LIN {X 0,Y 445.491,Z 467.925,A -85,B 0,C 180,E1 -8723.659,E2 -8723.659} C_VEL
LIN {X 0,Y 445.471,Z 472.126,A -85,B 0,C 180,E1 -8725.021,E2 -8725.021} C_VEL
LIN {X 0,Y 445.391,Z 475.228,A -85,B 0,C 180,E1 -8726.38,E2 -8726.38} C_VEL
LIN {X 0,Y 445.448,Z 476.703,A -85,B 0,C 180,E1 -8727.286,E2 -8727.286} C_VEL
LIN {X 0,Y 445.399,Z 477.757,A -85,B 0,C 180,E1 -8728.191,E2 -8728.191} C_VEL
LIN {X 0,Y 445.398,Z 478.402,A -85,B 0,C 180,E1 -8729.095,E2 -8729.095} C_VEL
LIN {X 0,Y 445.406,Z 478.591,A -85,B 0,C 180,E1 -8729.999,E2 -8729.999} C_VEL
LIN {X 0,Y 445.398,Z 478.345,A -85,B 0,C 180,E1 -8730.903,E2 -8730.903} C_VEL
LIN {X 0,Y 445.399,Z 477.688,A -85,B 0,C 180,E1 -8731.807,E2 -8731.807} C_VEL
LIN {X 0,Y 445.452,Z 476.615,A -85,B 0,C 180,E1 -8732.712,E2 -8732.712} C_VEL
LIN {X 0,Y 445.399,Z 474.132,A -85,B 0,C 180,E1 -8734.071,E2 -8734.071} C_VEL
LIN {X 0,Y 445.479,Z 470.6,A -85,B 0,C 180,E1 -8735.431,E2 -8735.431} C_VEL
LIN {X 0,Y 445.542,Z 465.911,A -85,B 0,C 180,E1 -8736.793,E2 -8736.793} C_VEL
LIN {X 0,Y 445.738,Z 459.918,A -85,B 0,C 180,E1 -8738.157,E2 -8738.157} C_VEL
LIN {X 0,Y 446.06,Z 449.817,A -85,B 0,C 180,E1 -8739.979,E2 -8739.979} C_VEL
LIN {X 0,Y 446.499,Z 442.125,A -85,B 0,C 180,E1 -8741.116,E2 -8741.116} C_VEL
LIN {X 0,Y 447.018,Z 432.751,A -85,B 0,C 180,E1 -8742.253,E2 -8742.253} C_VEL
LIN {X 0,Y 447.601,Z 421.509,A -85,B 0,C 180,E1 -8743.348,E2 -8743.348} C_VEL
LIN {X 0,Y 448.216,Z 410.725,A -85,B 0,C 180,E1 -8744.181,E2 -8744.181} C_VEL
LIN {X 0,Y 448.805,Z 398.322,A -85,B 0,C 180,E1 -8744.915,E2 -8744.915} C_VEL
LIN {X 0,Y 449.352,Z 385.98,A -85,B 0,C 180,E1 -8745.448,E2 -8745.448} C_VEL
LIN {X 0,Y 449.771,Z 373.319,A -85,B 0,C 180,E1 -8745.81,E2 -8745.81} C_VEL
LIN {X 0,Y 450.349,Z 287.235,A -85,B 0,C 180,E1 -8747.236,E2 -8747.236} C_VEL
LIN {X 0,Y 447.336,Z 266.21,A -85,B 0,C 180,E1 -8747.733,E2 -8747.733} C_VEL
LIN {X 0,Y 448.035,Z 250.938,A -85,B 0,C 180,E1 -8750.426,E2 -8750.426} C_VEL
LIN {X 0,Y 449,Z 233.588,A -85,B 0,C 180,E1 -8753.523,E2 -8753.523} C_VEL
LIN {X 0,Y 449.257,Z 228.525,A -85,B 0,C 180,E1 -8754.438,E2 -8754.438} C_VEL
LIN {X 0,Y 447.389,Z 218.203,A -85,B 0,C 180,E1 -8756.439,E2 -8756.439} C_VEL
LIN {X 0,Y 446.519,Z 213.866,A -85,B 0,C 180,E1 -8757.315,E2 -8757.315} C_VEL
LIN {X 0,Y 446.424,Z 213.878,A -85,B 0,C 180,E1 -8760.249,E2 -8760.249} C_VEL
LIN {X 0,Y 446.441,Z 213.856,A -85,B 0,C 180,E1 -8763.453,E2 -8763.453} C_VEL
LIN {X 0,Y 446.395,Z 213.877,A -85,B 0,C 180,E1 -8766.745,E2 -8766.745} C_VEL
LIN {X 0,Y 446.395,Z 213.875,A -85,B 0,C 180,E1 -8769.516,E2 -8769.516} C_VEL
LIN {X 0,Y 446.41,Z 213.872,A -85,B 0,C 180,E1 -8772.605,E2 -8772.605} C_VEL
LIN {X 0,Y 446.443,Z 213.872,A -85,B 0,C 180,E1 -8775.103,E2 -8775.103} C_VEL
LIN {X 0,Y 446.399,Z 213.867,A -85,B 0,C 180,E1 -8778.606,E2 -8778.606} C_VEL
LIN {X 0,Y 446.404,Z 213.875,A -85,B 0,C 180,E1 -8781.921,E2 -8781.921} C_VEL
LIN {X 0,Y 446.415,Z 213.873,A -85,B 0,C 180,E1 -8785.476,E2 -8785.476} C_VEL
LIN {X 0,Y 446.406,Z 213.874,A -85,B 0,C 180,E1 -8788.699,E2 -8788.699} C_VEL
LIN {X 0,Y 446.415,Z 213.866,A -85,B 0,C 180,E1 -8791.836,E2 -8791.836} C_VEL
LIN {X 0,Y 446.41,Z 213.877,A -85,B 0,C 180,E1 -8794.845,E2 -8794.845} C_VEL
LIN {X 0,Y 446.439,Z 213.854,A -85,B 0,C 180,E1 -8798.245,E2 -8798.245} C_VEL
LIN {X 0,Y 446.437,Z 213.87,A -85,B 0,C 180,E1 -8801.648,E2 -8801.648} C_VEL
LIN {X 0,Y 446.482,Z 213.862,A -85,B 0,C 180,E1 -8804.479,E2 -8804.479} C_VEL
LIN {X 0,Y 446.506,Z 213.858,A -85,B 0,C 180,E1 -8808.193,E2 -8808.193} C_VEL
LIN {X 0,Y 446.52,Z 213.863,A -85,B 0,C 180,E1 -8810.944,E2 -8810.944} C_VEL
LIN {X 0,Y 446.589,Z 213.843,A -85,B 0,C 180,E1 -8813.676,E2 -8813.676} C_VEL
LIN {X 0,Y 446.669,Z 213.839,A -85,B 0,C 180,E1 -8817.295,E2 -8817.295} C_VEL
LIN {X 0,Y 446.728,Z 213.837,A -85,B 0,C 180,E1 -8820,E2 -8820} C_VEL
LIN {X 0,Y 446.652,Z 213.83,A -85,B 0,C 180,E1 -8822.706,E2 -8822.706} C_VEL
LIN {X 0,Y 446.63,Z 213.849,A -85,B 0,C 180,E1 -8826.324,E2 -8826.324} C_VEL
LIN {X 0,Y 446.527,Z 213.851,A -85,B 0,C 180,E1 -8829.056,E2 -8829.056} C_VEL
LIN {X 0,Y 446.513,Z 213.859,A -85,B 0,C 180,E1 -8832.73,E2 -8832.73} C_VEL
LIN {X 0,Y 446.488,Z 213.858,A -85,B 0,C 180,E1 -8836.228,E2 -8836.228} C_VEL
LIN {X 0,Y 446.461,Z 213.866,A -85,B 0,C 180,E1 -8839.304,E2 -8839.304} C_VEL
LIN {X 0,Y 446.411,Z 213.872,A -85,B 0,C 180,E1 -8842.2,E2 -8842.2} C_VEL
LIN {X 0,Y 446.451,Z 213.867,A -85,B 0,C 180,E1 -8845.153,E2 -8845.153} C_VEL
LIN {X 0,Y 446.478,Z 213.863,A -85,B 0,C 180,E1 -8848.18,E2 -8848.18} C_VEL
LIN {X 0,Y 446.414,Z 213.878,A -85,B 0,C 180,E1 -8851.776,E2 -8851.776} C_VEL
LIN {X 0,Y 446.425,Z 213.869,A -85,B 0,C 180,E1 -8854.524,E2 -8854.524} C_VEL
LIN {X 0,Y 446.426,Z 213.87,A -85,B 0,C 180,E1 -8858.083,E2 -8858.083} C_VEL
LIN {X 0,Y 446.423,Z 213.881,A -85,B 0,C 180,E1 -8860.919,E2 -8860.919} C_VEL
LIN {X 0,Y 446.419,Z 213.875,A -85,B 0,C 180,E1 -8863.844,E2 -8863.844} C_VEL
LIN {X 0,Y 446.417,Z 213.877,A -85,B 0,C 180,E1 -8866.402,E2 -8866.402} C_VEL
LIN {X 0,Y 446.445,Z 213.87,A -85,B 0,C 180,E1 -8869.804,E2 -8869.804} C_VEL
LIN {X 0,Y 446.407,Z 213.876,A -85,B 0,C 180,E1 -8872.123,E2 -8872.123} C_VEL
LIN {X 0,Y 446.439,Z 213.875,A -85,B 0,C 180,E1 -8875.479,E2 -8875.479} C_VEL
LIN {X 0,Y 446.539,Z 213.996,A -85,B 0,C 180,E1 -8877.013,E2 -8877.013} C_VEL
LIN {X 0,Y 447.57,Z 218.946,A -85,B 0,C 180,E1 -8877.6,E2 -8877.6} C_VEL
LIN {X 0,Y 447.76,Z 222.768,A -85,B 0,C 180,E1 -8877.987,E2 -8877.987} C_VEL
LIN {X 0,Y 451.423,Z 242.555,A -85,B 0,C 180,E1 -8878.491,E2 -8878.491} C_VEL
LIN {X 0,Y 450.451,Z 334.568,A -85,B 0,C 180,E1 -8880.001,E2 -8880.001} C_VEL
LIN {X 0,Y 450.12,Z 347.295,A -85,B 0,C 180,E1 -8880.38,E2 -8880.38} C_VEL
LIN {X 0,Y 449.73,Z 360.095,A -85,B 0,C 180,E1 -8880.961,E2 -8880.961} C_VEL
LIN {X 0,Y 449.262,Z 371.242,A -85,B 0,C 180,E1 -8881.638,E2 -8881.638} C_VEL
LIN {X 0,Y 448.644,Z 382.135,A -85,B 0,C 180,E1 -8882.478,E2 -8882.478} C_VEL
LIN {X 0,Y 447.989,Z 392.819,A -85,B 0,C 180,E1 -8883.518,E2 -8883.518} C_VEL
LIN {X 0,Y 447.444,Z 402.256,A -85,B 0,C 180,E1 -8884.66,E2 -8884.66} C_VEL
LIN {X 0,Y 446.879,Z 410.422,A -85,B 0,C 180,E1 -8885.866,E2 -8885.866} C_VEL
LIN {X 0,Y 446.63,Z 415.074,A -85,B 0,C 180,E1 -8886.684,E2 -8886.684} C_VEL
LIN {X 0,Y 445.742,Z 418.376,A -85,B 0,C 180,E1 -8887.309,E2 -8887.309} C_VEL
LIN {X 0,Y 442.578,Z 423.342,A -85,B 0,C 180,E1 -8888.342,E2 -8888.342} C_VEL
LIN {X 0,Y 439.477,Z 427.618,A -85,B 0,C 180,E1 -8889.432,E2 -8889.432} C_VEL
LIN {X 0,Y 438.697,Z 429.804,A -85,B 0,C 180,E1 -8890.138,E2 -8890.138} C_VEL
LIN {X 0,Y 438.551,Z 432.748,A -85,B 0,C 180,E1 -8891.307,E2 -8891.307} C_VEL
LIN {X 0,Y 438.403,Z 434.652,A -85,B 0,C 180,E1 -8892.268,E2 -8892.268} C_VEL
LIN {X 0,Y 438.315,Z 436.052,A -85,B 0,C 180,E1 -8893.226,E2 -8893.226} C_VEL
LIN {X 0,Y 438.281,Z 437.025,A -85,B 0,C 180,E1 -8894.182,E2 -8894.182} C_VEL
LIN {X 0,Y 438.267,Z 437.592,A -85,B 0,C 180,E1 -8895.134,E2 -8895.134} C_VEL
LIN {X 0,Y 438.214,Z 437.705,A -85,B 0,C 180,E1 -8896.081,E2 -8896.081} C_VEL
LIN {X 0,Y 438.255,Z 437.402,A -85,B 0,C 180,E1 -8897.027,E2 -8897.027} C_VEL
LIN {X 0,Y 438.338,Z 436.705,A -85,B 0,C 180,E1 -8897.971,E2 -8897.971} C_VEL
LIN {X 0,Y 438.335,Z 435.586,A -85,B 0,C 180,E1 -8898.908,E2 -8898.908} C_VEL
LIN {X 0,Y 438.372,Z 434.026,A -85,B 0,C 180,E1 -8899.844,E2 -8899.844} C_VEL
LIN {X 0,Y 438.547,Z 430.873,A -85,B 0,C 180,E1 -8901.244,E2 -8901.244} C_VEL
LIN {X 0,Y 438.774,Z 426.656,A -85,B 0,C 180,E1 -8902.639,E2 -8902.639} C_VEL
LIN {X 0,Y 438.998,Z 421.278,A -85,B 0,C 180,E1 -8904.028,E2 -8904.028} C_VEL
LIN {X 0,Y 439.425,Z 414.546,A -85,B 0,C 180,E1 -8905.414,E2 -8905.414} C_VEL
LIN {X 0,Y 439.833,Z 406.138,A -85,B 0,C 180,E1 -8906.795,E2 -8906.795} C_VEL
LIN {X 0,Y 440.343,Z 397.532,A -85,B 0,C 180,E1 -8907.943,E2 -8907.943} C_VEL
LIN {X 0,Y 440.982,Z 386.969,A -85,B 0,C 180,E1 -8909.088,E2 -8909.088} C_VEL
LIN {X 0,Y 441.589,Z 376.354,A -85,B 0,C 180,E1 -8910.001,E2 -8910.001} C_VEL
LIN {X 0,Y 442.106,Z 364.638,A -85,B 0,C 180,E1 -8910.798,E2 -8910.798} C_VEL
LIN {X 0,Y 442.544,Z 352.502,A -85,B 0,C 180,E1 -8911.423,E2 -8911.423} C_VEL
LIN {X 0,Y 442.848,Z 339.912,A -85,B 0,C 180,E1 -8911.877,E2 -8911.877} C_VEL
LIN {X 0,Y 443.043,Z 326.53,A -85,B 0,C 180,E1 -8912.172,E2 -8912.172} C_VEL
LIN {X 0,Y 443.806,Z 242.883,A -85,B 0,C 180,E1 -8913.526,E2 -8913.526} C_VEL
LIN {X 0,Y 440.196,Z 222.44,A -85,B 0,C 180,E1 -8914.006,E2 -8914.006} C_VEL
LIN {X 0,Y 439.772,Z 216.284,A -85,B 0,C 180,E1 -8914.699,E2 -8914.699} C_VEL
LIN {X 0,Y 439.485,Z 214.744,A -85,B 0,C 180,E1 -8914.903,E2 -8914.903} C_VEL
LIN {X 0,Y 439.58,Z 214.732,A -85,B 0,C 180,E1 -8917.579,E2 -8917.579} C_VEL
LIN {X 0,Y 439.438,Z 214.748,A -85,B 0,C 180,E1 -8921.066,E2 -8921.066} C_VEL
LIN {X 0,Y 439.425,Z 214.749,A -85,B 0,C 180,E1 -8923.882,E2 -8923.882} C_VEL
LIN {X 0,Y 439.454,Z 214.747,A -85,B 0,C 180,E1 -8926.731,E2 -8926.731} C_VEL
LIN {X 0,Y 439.409,Z 214.751,A -85,B 0,C 180,E1 -8929.627,E2 -8929.627} C_VEL
LIN {X 0,Y 439.369,Z 214.758,A -85,B 0,C 180,E1 -8932.576,E2 -8932.576} C_VEL
LIN {X 0,Y 439.372,Z 214.755,A -85,B 0,C 180,E1 -8935.588,E2 -8935.588} C_VEL
LIN {X 0,Y 439.396,Z 214.752,A -85,B 0,C 180,E1 -8938.676,E2 -8938.676} C_VEL
LIN {X 0,Y 439.369,Z 214.756,A -85,B 0,C 180,E1 -8942.029,E2 -8942.029} C_VEL
LIN {X 0,Y 439.395,Z 214.752,A -85,B 0,C 180,E1 -8945.34,E2 -8945.34} C_VEL
LIN {X 0,Y 439.355,Z 214.757,A -85,B 0,C 180,E1 -8948.599,E2 -8948.599} C_VEL
LIN {X 0,Y 439.35,Z 214.758,A -85,B 0,C 180,E1 -8952.211,E2 -8952.211} C_VEL
LIN {X 0,Y 439.377,Z 214.754,A -85,B 0,C 180,E1 -8955.267,E2 -8955.267} C_VEL
LIN {X 0,Y 439.363,Z 214.757,A -85,B 0,C 180,E1 -8958.748,E2 -8958.748} C_VEL
LIN {X 0,Y 439.355,Z 214.759,A -85,B 0,C 180,E1 -8961.612,E2 -8961.612} C_VEL
LIN {X 0,Y 439.356,Z 214.757,A -85,B 0,C 180,E1 -8964.84,E2 -8964.84} C_VEL
LIN {X 0,Y 439.352,Z 214.757,A -85,B 0,C 180,E1 -8968.137,E2 -8968.137} C_VEL
LIN {X 0,Y 439.383,Z 214.755,A -85,B 0,C 180,E1 -8971.324,E2 -8971.324} C_VEL
LIN {X 0,Y 439.36,Z 214.757,A -85,B 0,C 180,E1 -8974.412,E2 -8974.412} C_VEL
LIN {X 0,Y 439.371,Z 214.758,A -85,B 0,C 180,E1 -8977.424,E2 -8977.424} C_VEL
LIN {X 0,Y 439.442,Z 214.849,A -85,B 0,C 180,E1 -8978.241,E2 -8978.241} C_VEL
LIN {X 0,Y 440.59,Z 221.732,A -85,B 0,C 180,E1 -8979.914,E2 -8979.914} C_VEL
LIN {X 0,Y 440.519,Z 227.273,A -85,B 0,C 180,E1 -8981.2,E2 -8981.2} C_VEL
LIN {X 0,Y 443.718,Z 244.798,A -85,B 0,C 180,E1 -8981.663,E2 -8981.663} C_VEL
LIN {X 0,Y 442.305,Z 335.472,A -85,B 0,C 180,E1 -8983.41,E2 -8983.41} C_VEL
LIN {X 0,Y 442.029,Z 348.552,A -85,B 0,C 180,E1 -8983.845,E2 -8983.845} C_VEL
LIN {X 0,Y 441.695,Z 360.749,A -85,B 0,C 180,E1 -8984.424,E2 -8984.424} C_VEL
LIN {X 0,Y 441.149,Z 373.393,A -85,B 0,C 180,E1 -8985.232,E2 -8985.232} C_VEL
LIN {X 0,Y 440.66,Z 384.739,A -85,B 0,C 180,E1 -8986.158,E2 -8986.158} C_VEL
LIN {X 0,Y 440.198,Z 394.951,A -85,B 0,C 180,E1 -8987.201,E2 -8987.201} C_VEL
LIN {X 0,Y 439.742,Z 405.029,A -85,B 0,C 180,E1 -8988.476,E2 -8988.476} C_VEL
LIN {X 0,Y 439.344,Z 412.509,A -85,B 0,C 180,E1 -8989.632,E2 -8989.632} C_VEL
LIN {X 0,Y 439.028,Z 419.839,A -85,B 0,C 180,E1 -8991.02,E2 -8991.02} C_VEL
LIN {X 0,Y 438.713,Z 426.499,A -85,B 0,C 180,E1 -8992.637,E2 -8992.637} C_VEL
LIN {X 0,Y 438.619,Z 430.873,A -85,B 0,C 180,E1 -8994.022,E2 -8994.022} C_VEL
LIN {X 0,Y 438.43,Z 434.134,A -85,B 0,C 180,E1 -8995.403,E2 -8995.403} C_VEL
LIN {X 0,Y 438.475,Z 435.757,A -85,B 0,C 180,E1 -8996.324,E2 -8996.324} C_VEL
LIN {X 0,Y 438.437,Z 436.903,A -85,B 0,C 180,E1 -8997.243,E2 -8997.243} C_VEL
LIN {X 0,Y 438.353,Z 437.639,A -85,B 0,C 180,E1 -8998.162,E2 -8998.162} C_VEL
LIN {X 0,Y 438.329,Z 437.972,A -85,B 0,C 180,E1 -8999.081,E2 -8999.081} C_VEL
LIN {X 0,Y 438.351,Z 437.874,A -85,B 0,C 180,E1 -9000,E2 -9000} C_VEL
LIN {X 0,Y 438.381,Z 437.328,A -85,B 0,C 180,E1 -9000.918,E2 -9000.918} C_VEL
LIN {X 0,Y 438.464,Z 436.376,A -85,B 0,C 180,E1 -9001.837,E2 -9001.837} C_VEL
LIN {X 0,Y 438.596,Z 435.012,A -85,B 0,C 180,E1 -9002.755,E2 -9002.755} C_VEL
LIN {X 0,Y 438.716,Z 432.097,A -85,B 0,C 180,E1 -9004.134,E2 -9004.134} C_VEL
LIN {X 0,Y 438.801,Z 428.123,A -85,B 0,C 180,E1 -9005.514,E2 -9005.514} C_VEL
LIN {X 0,Y 439.197,Z 422.959,A -85,B 0,C 180,E1 -9006.889,E2 -9006.889} C_VEL
LIN {X 0,Y 439.52,Z 416.402,A -85,B 0,C 180,E1 -9008.274,E2 -9008.274} C_VEL
LIN {X 0,Y 440.047,Z 408.237,A -85,B 0,C 180,E1 -9009.654,E2 -9009.654} C_VEL
LIN {X 0,Y 440.481,Z 399.912,A -85,B 0,C 180,E1 -9010.805,E2 -9010.805} C_VEL
LIN {X 0,Y 441.02,Z 389.655,A -85,B 0,C 180,E1 -9011.956,E2 -9011.956} C_VEL
LIN {X 0,Y 441.787,Z 378.093,A -85,B 0,C 180,E1 -9012.985,E2 -9012.985} C_VEL
LIN {X 0,Y 442.249,Z 366.753,A -85,B 0,C 180,E1 -9013.79,E2 -9013.79} C_VEL
LIN {X 0,Y 442.792,Z 353.746,A -85,B 0,C 180,E1 -9014.487,E2 -9014.487} C_VEL
LIN {X 0,Y 443.124,Z 340.608,A -85,B 0,C 180,E1 -9014.994,E2 -9014.994} C_VEL
LIN {X 0,Y 443.464,Z 323.313,A -85,B 0,C 180,E1 -9015.394,E2 -9015.394} C_VEL
LIN {X 0,Y 445.269,Z 245.911,A -85,B 0,C 180,E1 -9017.013,E2 -9017.013} C_VEL
LIN {X 0,Y 442.888,Z 234.755,A -85,B 0,C 180,E1 -9017.414,E2 -9017.414} C_VEL
LIN {X 0,Y 441.713,Z 230.459,A -85,B 0,C 180,E1 -9017.596,E2 -9017.596} C_VEL
LIN {X 0,Y 441.551,Z 225.043,A -85,B 0,C 180,E1 -9019.044,E2 -9019.044} C_VEL
LIN {X 0,Y 440.169,Z 218.137,A -85,B 0,C 180,E1 -9021.054,E2 -9021.054} C_VEL
LIN {X 0,Y 439.396,Z 214.755,A -85,B 0,C 180,E1 -9022.135,E2 -9022.135} C_VEL
LIN {X 0,Y 439.415,Z 214.754,A -85,B 0,C 180,E1 -9024.572,E2 -9024.572} C_VEL
LIN {X 0,Y 439.446,Z 214.747,A -85,B 0,C 180,E1 -9027.632,E2 -9027.632} C_VEL
LIN {X 0,Y 439.366,Z 214.756,A -85,B 0,C 180,E1 -9030.788,E2 -9030.788} C_VEL
LIN {X 0,Y 439.393,Z 214.754,A -85,B 0,C 180,E1 -9034.043,E2 -9034.043} C_VEL
LIN {X 0,Y 439.353,Z 214.757,A -85,B 0,C 180,E1 -9036.887,E2 -9036.887} C_VEL
LIN {X 0,Y 439.407,Z 214.751,A -85,B 0,C 180,E1 -9039.849,E2 -9039.849} C_VEL
LIN {X 0,Y 439.386,Z 214.755,A -85,B 0,C 180,E1 -9042.626,E2 -9042.626} C_VEL
LIN {X 0,Y 439.404,Z 214.75,A -85,B 0,C 180,E1 -9045.27,E2 -9045.27} C_VEL
LIN {X 0,Y 439.386,Z 214.753,A -85,B 0,C 180,E1 -9048.744,E2 -9048.744} C_VEL
LIN {X 0,Y 439.372,Z 214.756,A -85,B 0,C 180,E1 -9051.608,E2 -9051.608} C_VEL
LIN {X 0,Y 439.403,Z 214.752,A -85,B 0,C 180,E1 -9054.843,E2 -9054.843} C_VEL
LIN {X 0,Y 439.378,Z 214.761,A -85,B 0,C 180,E1 -9058.139,E2 -9058.139} C_VEL
LIN {X 0,Y 439.461,Z 214.832,A -85,B 0,C 180,E1 -9061.296,E2 -9061.296} C_VEL
LIN {X 0,Y 441.873,Z 225.21,A -85,B 0,C 180,E1 -9063.808,E2 -9063.808} C_VEL
LIN {X 0,Y 442.962,Z 231.622,A -85,B 0,C 180,E1 -9065.228,E2 -9065.228} C_VEL
LIN {X 0,Y 441.856,Z 246.026,A -85,B 0,C 180,E1 -9068.05,E2 -9068.05} C_VEL
LIN {X 0,Y 440.748,Z 263.778,A -85,B 0,C 180,E1 -9071.372,E2 -9071.372} C_VEL
LIN {X 0,Y 443.807,Z 282.169,A -85,B 0,C 180,E1 -9071.969,E2 -9071.969} C_VEL
LIN {X 0,Y 444.568,Z 290.239,A -85,B 0,C 180,E1 -9072.193,E2 -9072.193} C_VEL
LIN {X 0,Y 442.911,Z 375.135,A -85,B 0,C 180,E1 -9073.966,E2 -9073.966} C_VEL
LIN {X 0,Y 442.448,Z 387.688,A -85,B 0,C 180,E1 -9074.392,E2 -9074.392} C_VEL
LIN {X 0,Y 441.859,Z 399.713,A -85,B 0,C 180,E1 -9074.961,E2 -9074.961} C_VEL
LIN {X 0,Y 441.212,Z 411.543,A -85,B 0,C 180,E1 -9075.705,E2 -9075.705} C_VEL
LIN {X 0,Y 440.53,Z 423.87,A -85,B 0,C 180,E1 -9076.697,E2 -9076.697} C_VEL
LIN {X 0,Y 439.914,Z 434.527,A -85,B 0,C 180,E1 -9077.778,E2 -9077.778} C_VEL
LIN {X 0,Y 439.427,Z 443.816,A -85,B 0,C 180,E1 -9078.934,E2 -9078.934} C_VEL
LIN {X 0,Y 438.957,Z 452.908,A -85,B 0,C 180,E1 -9080.321,E2 -9080.321} C_VEL
LIN {X 0,Y 438.663,Z 460.162,A -85,B 0,C 180,E1 -9081.708,E2 -9081.708} C_VEL
LIN {X 0,Y 438.458,Z 465.984,A -85,B 0,C 180,E1 -9083.094,E2 -9083.094} C_VEL
LIN {X 0,Y 438.363,Z 470.556,A -85,B 0,C 180,E1 -9084.479,E2 -9084.479} C_VEL
LIN {X 0,Y 438.346,Z 472.986,A -85,B 0,C 180,E1 -9085.401,E2 -9085.401} C_VEL
LIN {X 0,Y 438.292,Z 474.931,A -85,B 0,C 180,E1 -9086.322,E2 -9086.322} C_VEL
LIN {X 0,Y 438.373,Z 476.401,A -85,B 0,C 180,E1 -9087.242,E2 -9087.242} C_VEL
LIN {X 0,Y 438.318,Z 477.447,A -85,B 0,C 180,E1 -9088.161,E2 -9088.161} C_VEL
LIN {X 0,Y 438.308,Z 478.08,A -85,B 0,C 180,E1 -9089.08,E2 -9089.08} C_VEL
LIN {X 0,Y 438.327,Z 478.247,A -85,B 0,C 180,E1 -9089.999,E2 -9089.999} C_VEL
LIN {X 0,Y 438.308,Z 477.987,A -85,B 0,C 180,E1 -9090.918,E2 -9090.918} C_VEL
LIN {X 0,Y 438.319,Z 477.316,A -85,B 0,C 180,E1 -9091.837,E2 -9091.837} C_VEL
LIN {X 0,Y 438.378,Z 476.214,A -85,B 0,C 180,E1 -9092.756,E2 -9092.756} C_VEL
LIN {X 0,Y 438.31,Z 473.696,A -85,B 0,C 180,E1 -9094.137,E2 -9094.137} C_VEL
LIN {X 0,Y 438.374,Z 470.118,A -85,B 0,C 180,E1 -9095.519,E2 -9095.519} C_VEL
LIN {X 0,Y 438.462,Z 465.369,A -85,B 0,C 180,E1 -9096.903,E2 -9096.903} C_VEL
LIN {X 0,Y 438.693,Z 458.257,A -85,B 0,C 180,E1 -9098.521,E2 -9098.521} C_VEL
LIN {X 0,Y 438.996,Z 451.021,A -85,B 0,C 180,E1 -9099.909,E2 -9099.909} C_VEL
LIN {X 0,Y 439.517,Z 442.02,A -85,B 0,C 180,E1 -9101.295,E2 -9101.295} C_VEL
LIN {X 0,Y 440.063,Z 432.715,A -85,B 0,C 180,E1 -9102.45,E2 -9102.45} C_VEL
LIN {X 0,Y 440.659,Z 421.888,A -85,B 0,C 180,E1 -9103.531,E2 -9103.531} C_VEL
LIN {X 0,Y 441.35,Z 410.866,A -85,B 0,C 180,E1 -9104.406,E2 -9104.406} C_VEL
LIN {X 0,Y 441.967,Z 398.672,A -85,B 0,C 180,E1 -9105.151,E2 -9105.151} C_VEL
LIN {X 0,Y 442.547,Z 385.833,A -85,B 0,C 180,E1 -9105.721,E2 -9105.721} C_VEL
LIN {X 0,Y 443.019,Z 373.335,A -85,B 0,C 180,E1 -9106.087,E2 -9106.087} C_VEL
LIN {X 0,Y 443.735,Z 288.571,A -85,B 0,C 180,E1 -9107.512,E2 -9107.512} C_VEL
LIN {X 0,Y 440.393,Z 265.376,A -85,B 0,C 180,E1 -9108.082,E2 -9108.082} C_VEL
LIN {X 0,Y 441.318,Z 246.448,A -85,B 0,C 180,E1 -9111.485,E2 -9111.485} C_VEL
LIN {X 0,Y 442.308,Z 230.434,A -85,B 0,C 180,E1 -9114.4,E2 -9114.4} C_VEL
LIN {X 0,Y 441.275,Z 223.616,A -85,B 0,C 180,E1 -9115.72,E2 -9115.72} C_VEL
LIN {X 0,Y 439.496,Z 214.742,A -85,B 0,C 180,E1 -9117.498,E2 -9117.498} C_VEL
LIN {X 0,Y 439.358,Z 214.755,A -85,B 0,C 180,E1 -9120.787,E2 -9120.787} C_VEL
LIN {X 0,Y 439.383,Z 214.735,A -85,B 0,C 180,E1 -9124.043,E2 -9124.043} C_VEL
LIN {X 0,Y 439.341,Z 214.756,A -85,B 0,C 180,E1 -9126.886,E2 -9126.886} C_VEL
LIN {X 0,Y 439.342,Z 214.757,A -85,B 0,C 180,E1 -9129.84,E2 -9129.84} C_VEL
LIN {X 0,Y 439.363,Z 214.749,A -85,B 0,C 180,E1 -9132.624,E2 -9132.624} C_VEL
LIN {X 0,Y 439.391,Z 214.752,A -85,B 0,C 180,E1 -9135.269,E2 -9135.269} C_VEL
LIN {X 0,Y 439.349,Z 214.747,A -85,B 0,C 180,E1 -9139.016,E2 -9139.016} C_VEL
LIN {X 0,Y 439.339,Z 214.753,A -85,B 0,C 180,E1 -9142.564,E2 -9142.564} C_VEL
LIN {X 0,Y 439.388,Z 214.739,A -85,B 0,C 180,E1 -9144.843,E2 -9144.843} C_VEL
LIN {X 0,Y 439.363,Z 214.75,A -85,B 0,C 180,E1 -9148.139,E2 -9148.139} C_VEL
LIN {X 0,Y 439.391,Z 214.742,A -85,B 0,C 180,E1 -9151.606,E2 -9151.606} C_VEL
LIN {X 0,Y 439.356,Z 214.752,A -85,B 0,C 180,E1 -9154.412,E2 -9154.412} C_VEL
LIN {X 0,Y 439.352,Z 214.737,A -85,B 0,C 180,E1 -9157.424,E2 -9157.424} C_VEL
LIN {X 0,Y 439.431,Z 214.743,A -85,B 0,C 180,E1 -9160.663,E2 -9160.663} C_VEL
LIN {X 0,Y 439.443,Z 214.74,A -85,B 0,C 180,E1 -9164.224,E2 -9164.224} C_VEL
LIN {X 0,Y 439.473,Z 214.732,A -85,B 0,C 180,E1 -9168.001,E2 -9168.001} C_VEL
LIN {X 0,Y 439.493,Z 214.735,A -85,B 0,C 180,E1 -9171.725,E2 -9171.725} C_VEL
LIN {X 0,Y 439.582,Z 214.712,A -85,B 0,C 180,E1 -9174.495,E2 -9174.495} C_VEL
LIN {X 0,Y 439.623,Z 214.722,A -85,B 0,C 180,E1 -9178.168,E2 -9178.168} C_VEL
LIN {X 0,Y 439.587,Z 214.717,A -85,B 0,C 180,E1 -9180.916,E2 -9180.916} C_VEL
LIN {X 0,Y 439.604,Z 214.707,A -85,B 0,C 180,E1 -9182.749,E2 -9182.749} C_VEL
LIN {X 0,Y 439.602,Z 214.723,A -85,B 0,C 180,E1 -9186.426,E2 -9186.426} C_VEL
LIN {X 0,Y 439.489,Z 214.728,A -85,B 0,C 180,E1 -9189.202,E2 -9189.202} C_VEL
LIN {X 0,Y 439.457,Z 214.737,A -85,B 0,C 180,E1 -9192.938,E2 -9192.938} C_VEL
LIN {X 0,Y 439.438,Z 214.734,A -85,B 0,C 180,E1 -9196.349,E2 -9196.349} C_VEL
LIN {X 0,Y 439.394,Z 214.75,A -85,B 0,C 180,E1 -9199.627,E2 -9199.627} C_VEL
LIN {X 0,Y 439.358,Z 214.749,A -85,B 0,C 180,E1 -9202.576,E2 -9202.576} C_VEL
LIN {X 0,Y 439.399,Z 214.751,A -85,B 0,C 180,E1 -9205.586,E2 -9205.586} C_VEL
LIN {X 0,Y 439.411,Z 214.743,A -85,B 0,C 180,E1 -9208.674,E2 -9208.674} C_VEL
LIN {X 0,Y 439.364,Z 214.754,A -85,B 0,C 180,E1 -9212.031,E2 -9212.031} C_VEL
LIN {X 0,Y 439.391,Z 214.754,A -85,B 0,C 180,E1 -9215.342,E2 -9215.342} C_VEL
LIN {X 0,Y 439.386,Z 214.748,A -85,B 0,C 180,E1 -9218.595,E2 -9218.595} C_VEL
LIN {X 0,Y 439.384,Z 214.752,A -85,B 0,C 180,E1 -9221.258,E2 -9221.258} C_VEL
LIN {X 0,Y 439.402,Z 214.751,A -85,B 0,C 180,E1 -9224.73,E2 -9224.73} C_VEL
LIN {X 0,Y 439.394,Z 214.749,A -85,B 0,C 180,E1 -9227.797,E2 -9227.797} C_VEL
LIN {X 0,Y 439.427,Z 214.745,A -85,B 0,C 180,E1 -9230.229,E2 -9230.229} C_VEL
LIN {X 0,Y 439.372,Z 214.754,A -85,B 0,C 180,E1 -9233.714,E2 -9233.714} C_VEL
LIN {X 0,Y 439.473,Z 214.811,A -85,B 0,C 180,E1 -9236.754,E2 -9236.754} C_VEL
LIN {X 0,Y 440.679,Z 219.63,A -85,B 0,C 180,E1 -9237.329,E2 -9237.329} C_VEL
LIN {X 0,Y 440.904,Z 222.871,A -85,B 0,C 180,E1 -9237.653,E2 -9237.653} C_VEL
LIN {X 0,Y 444.783,Z 243.787,A -85,B 0,C 180,E1 -9238.2,E2 -9238.2} C_VEL
LIN {X 0,Y 443.732,Z 334.723,A -85,B 0,C 180,E1 -9239.713,E2 -9239.713} C_VEL
LIN {X 0,Y 443.373,Z 347.934,A -85,B 0,C 180,E1 -9240.112,E2 -9240.112} C_VEL
LIN {X 0,Y 442.979,Z 359.967,A -85,B 0,C 180,E1 -9240.665,E2 -9240.665} C_VEL
LIN {X 0,Y 442.43,Z 372.414,A -85,B 0,C 180,E1 -9241.437,E2 -9241.437} C_VEL
LIN {X 0,Y 441.787,Z 382.926,A -85,B 0,C 180,E1 -9242.271,E2 -9242.271} C_VEL
LIN {X 0,Y 441.056,Z 393.927,A -85,B 0,C 180,E1 -9243.375,E2 -9243.375} C_VEL
LIN {X 0,Y 440.514,Z 402.858,A -85,B 0,C 180,E1 -9244.485,E2 -9244.485} C_VEL
LIN {X 0,Y 439.924,Z 410.846,A -85,B 0,C 180,E1 -9245.69,E2 -9245.69} C_VEL
LIN {X 0,Y 439.389,Z 418.76,A -85,B 0,C 180,E1 -9247.179,E2 -9247.179} C_VEL
LIN {X 0,Y 439.063,Z 424.005,A -85,B 0,C 180,E1 -9248.399,E2 -9248.399} C_VEL
LIN {X 0,Y 438.743,Z 428.993,A -85,B 0,C 180,E1 -9249.856,E2 -9249.856} C_VEL
LIN {X 0,Y 438.697,Z 429.804,A -85,B 0,C 180,E1 -9250.138,E2 -9250.138} C_VEL
LIN {X 0,Y 437.915,Z 431.79,A -85,B 0,C 180,E1 -9250.859,E2 -9250.859} C_VEL
LIN {X 0,Y 434.849,Z 434.5,A -85,B 0,C 180,E1 -9252.045,E2 -9252.045} C_VEL
LIN {X 0,Y 431.858,Z 436.49,A -85,B 0,C 180,E1 -9253.271,E2 -9253.271} C_VEL
LIN {X 0,Y 431.207,Z 437.279,A -85,B 0,C 180,E1 -9254.045,E2 -9254.045} C_VEL
LIN {X 0,Y 431.126,Z 438.043,A -85,B 0,C 180,E1 -9255.848,E2 -9255.848} C_VEL
LIN {X 0,Y 431.171,Z 437.819,A -85,B 0,C 180,E1 -9256.81,E2 -9256.81} C_VEL
LIN {X 0,Y 431.236,Z 437.064,A -85,B 0,C 180,E1 -9257.918,E2 -9257.918} C_VEL
LIN {X 0,Y 431.289,Z 434.711,A -85,B 0,C 180,E1 -9259.675,E2 -9259.675} C_VEL
LIN {X 0,Y 431.443,Z 431.702,A -85,B 0,C 180,E1 -9261.099,E2 -9261.099} C_VEL
LIN {X 0,Y 431.689,Z 427.631,A -85,B 0,C 180,E1 -9262.518,E2 -9262.518} C_VEL
LIN {X 0,Y 431.92,Z 422.409,A -85,B 0,C 180,E1 -9263.93,E2 -9263.93} C_VEL
LIN {X 0,Y 432.306,Z 415.858,A -85,B 0,C 180,E1 -9265.339,E2 -9265.339} C_VEL
LIN {X 0,Y 432.751,Z 407.745,A -85,B 0,C 180,E1 -9266.743,E2 -9266.743} C_VEL
LIN {X 0,Y 433.275,Z 399.383,A -85,B 0,C 180,E1 -9267.909,E2 -9267.909} C_VEL
LIN {X 0,Y 433.871,Z 389.153,A -85,B 0,C 180,E1 -9269.073,E2 -9269.073} C_VEL
LIN {X 0,Y 434.514,Z 379.034,A -85,B 0,C 180,E1 -9270.001,E2 -9270.001} C_VEL
LIN {X 0,Y 435.09,Z 367.953,A -85,B 0,C 180,E1 -9270.811,E2 -9270.811} C_VEL
LIN {X 0,Y 435.52,Z 355.564,A -85,B 0,C 180,E1 -9271.504,E2 -9271.504} C_VEL
LIN {X 0,Y 435.93,Z 342.606,A -85,B 0,C 180,E1 -9272.022,E2 -9272.022} C_VEL
LIN {X 0,Y 436.124,Z 329.95,A -85,B 0,C 180,E1 -9272.339,E2 -9272.339} C_VEL
LIN {X 0,Y 437,Z 243.946,A -85,B 0,C 180,E1 -9273.754,E2 -9273.754} C_VEL
LIN {X 0,Y 433.265,Z 222.529,A -85,B 0,C 180,E1 -9274.269,E2 -9274.269} C_VEL
LIN {X 0,Y 432.729,Z 216.946,A -85,B 0,C 180,E1 -9274.892,E2 -9274.892} C_VEL
LIN {X 0,Y 432.481,Z 215.618,A -85,B 0,C 180,E1 -9275.07,E2 -9275.07} C_VEL
LIN {X 0,Y 432.545,Z 215.608,A -85,B 0,C 180,E1 -9277.633,E2 -9277.633} C_VEL
LIN {X 0,Y 432.394,Z 215.624,A -85,B 0,C 180,E1 -9281.248,E2 -9281.248} C_VEL
LIN {X 0,Y 432.376,Z 215.626,A -85,B 0,C 180,E1 -9284.113,E2 -9284.113} C_VEL
LIN {X 0,Y 432.401,Z 215.624,A -85,B 0,C 180,E1 -9287.012,E2 -9287.012} C_VEL
LIN {X 0,Y 432.345,Z 215.63,A -85,B 0,C 180,E1 -9289.961,E2 -9289.961} C_VEL
LIN {X 0,Y 432.317,Z 215.633,A -85,B 0,C 180,E1 -9292.965,E2 -9292.965} C_VEL
LIN {X 0,Y 432.323,Z 215.633,A -85,B 0,C 180,E1 -9296.036,E2 -9296.036} C_VEL
LIN {X 0,Y 432.332,Z 215.632,A -85,B 0,C 180,E1 -9299.189,E2 -9299.189} C_VEL
LIN {X 0,Y 432.326,Z 215.633,A -85,B 0,C 180,E1 -9302.444,E2 -9302.444} C_VEL
LIN {X 0,Y 432.341,Z 215.631,A -85,B 0,C 180,E1 -9305.819,E2 -9305.819} C_VEL
LIN {X 0,Y 432.319,Z 215.633,A -85,B 0,C 180,E1 -9308.71,E2 -9308.71} C_VEL
LIN {X 0,Y 432.306,Z 215.636,A -85,B 0,C 180,E1 -9311.801,E2 -9311.801} C_VEL
LIN {X 0,Y 432.337,Z 215.631,A -85,B 0,C 180,E1 -9314.348,E2 -9314.348} C_VEL
LIN {X 0,Y 432.306,Z 215.636,A -85,B 0,C 180,E1 -9317.019,E2 -9317.019} C_VEL
LIN {X 0,Y 432.293,Z 215.638,A -85,B 0,C 180,E1 -9319.828,E2 -9319.828} C_VEL
LIN {X 0,Y 432.293,Z 215.637,A -85,B 0,C 180,E1 -9323.02,E2 -9323.02} C_VEL
LIN {X 0,Y 432.326,Z 215.632,A -85,B 0,C 180,E1 -9326.005,E2 -9326.005} C_VEL
LIN {X 0,Y 432.337,Z 215.632,A -85,B 0,C 180,E1 -9329.494,E2 -9329.494} C_VEL
LIN {X 0,Y 432.318,Z 215.633,A -85,B 0,C 180,E1 -9331.872,E2 -9331.872} C_VEL
LIN {X 0,Y 432.354,Z 215.629,A -85,B 0,C 180,E1 -9335.547,E2 -9335.547} C_VEL
LIN {X 0,Y 432.399,Z 215.8,A -85,B 0,C 180,E1 -9338.11,E2 -9338.11} C_VEL
LIN {X 0,Y 433.477,Z 221.813,A -85,B 0,C 180,E1 -9339.6,E2 -9339.6} C_VEL
LIN {X 0,Y 433.556,Z 227.515,A -85,B 0,C 180,E1 -9340.948,E2 -9340.948} C_VEL
LIN {X 0,Y 436.843,Z 245.736,A -85,B 0,C 180,E1 -9341.447,E2 -9341.447} C_VEL
LIN {X 0,Y 435.352,Z 335.791,A -85,B 0,C 180,E1 -9343.228,E2 -9343.228} C_VEL
LIN {X 0,Y 435.065,Z 349.571,A -85,B 0,C 180,E1 -9343.699,E2 -9343.699} C_VEL
LIN {X 0,Y 434.717,Z 361.528,A -85,B 0,C 180,E1 -9344.288,E2 -9344.288} C_VEL
LIN {X 0,Y 434.146,Z 374.07,A -85,B 0,C 180,E1 -9345.108,E2 -9345.108} C_VEL
LIN {X 0,Y 433.642,Z 385.352,A -85,B 0,C 180,E1 -9346.05,E2 -9346.05} C_VEL
LIN {X 0,Y 433.165,Z 395.502,A -85,B 0,C 180,E1 -9347.109,E2 -9347.109} C_VEL
LIN {X 0,Y 432.726,Z 404.717,A -85,B 0,C 180,E1 -9348.286,E2 -9348.286} C_VEL
LIN {X 0,Y 432.307,Z 412.314,A -85,B 0,C 180,E1 -9349.462,E2 -9349.462} C_VEL
LIN {X 0,Y 431.987,Z 419.774,A -85,B 0,C 180,E1 -9350.873,E2 -9350.873} C_VEL
LIN {X 0,Y 431.728,Z 424.793,A -85,B 0,C 180,E1 -9352.046,E2 -9352.046} C_VEL
LIN {X 0,Y 431.527,Z 429.656,A -85,B 0,C 180,E1 -9353.454,E2 -9353.454} C_VEL
LIN {X 0,Y 431.432,Z 433.348,A -85,B 0,C 180,E1 -9354.859,E2 -9354.859} C_VEL
LIN {X 0,Y 431.377,Z 435.979,A -85,B 0,C 180,E1 -9356.263,E2 -9356.263} C_VEL
LIN {X 0,Y 431.367,Z 437.175,A -85,B 0,C 180,E1 -9357.198,E2 -9357.198} C_VEL
LIN {X 0,Y 431.275,Z 437.94,A -85,B 0,C 180,E1 -9358.132,E2 -9358.132} C_VEL
LIN {X 0,Y 431.242,Z 438.3,A -85,B 0,C 180,E1 -9359.066,E2 -9359.066} C_VEL
LIN {X 0,Y 431.273,Z 438.246,A -85,B 0,C 180,E1 -9360,E2 -9360} C_VEL
LIN {X 0,Y 431.322,Z 437.729,A -85,B 0,C 180,E1 -9360.933,E2 -9360.933} C_VEL
LIN {X 0,Y 431.382,Z 436.804,A -85,B 0,C 180,E1 -9361.867,E2 -9361.867} C_VEL
LIN {X 0,Y 431.519,Z 435.465,A -85,B 0,C 180,E1 -9362.8,E2 -9362.8} C_VEL
LIN {X 0,Y 431.668,Z 432.594,A -85,B 0,C 180,E1 -9364.201,E2 -9364.201} C_VEL
LIN {X 0,Y 431.749,Z 428.662,A -85,B 0,C 180,E1 -9365.605,E2 -9365.605} C_VEL
LIN {X 0,Y 432.161,Z 423.822,A -85,B 0,C 180,E1 -9366.935,E2 -9366.935} C_VEL
LIN {X 0,Y 432.543,Z 417.068,A -85,B 0,C 180,E1 -9368.409,E2 -9368.409} C_VEL
LIN {X 0,Y 433.099,Z 408.966,A -85,B 0,C 180,E1 -9369.81,E2 -9369.81} C_VEL
LIN {X 0,Y 433.56,Z 400.709,A -85,B 0,C 180,E1 -9370.98,E2 -9370.98} C_VEL
LIN {X 0,Y 434.139,Z 390.597,A -85,B 0,C 180,E1 -9372.149,E2 -9372.149} C_VEL
LIN {X 0,Y 434.951,Z 379.175,A -85,B 0,C 180,E1 -9373.193,E2 -9373.193} C_VEL
LIN {X 0,Y 435.447,Z 368.058,A -85,B 0,C 180,E1 -9374.01,E2 -9374.01} C_VEL
LIN {X 0,Y 435.97,Z 356.708,A -85,B 0,C 180,E1 -9374.656,E2 -9374.656} C_VEL
LIN {X 0,Y 436.341,Z 343.751,A -85,B 0,C 180,E1 -9375.203,E2 -9375.203} C_VEL
LIN {X 0,Y 436.667,Z 329.967,A -85,B 0,C 180,E1 -9375.58,E2 -9375.58} C_VEL
LIN {X 0,Y 438.591,Z 252.836,A -85,B 0,C 180,E1 -9377.235,E2 -9377.235} C_VEL
LIN {X 0,Y 438.667,Z 245.788,A -85,B 0,C 180,E1 -9377.4,E2 -9377.4} C_VEL
LIN {X 0,Y 435.548,Z 233.175,A -85,B 0,C 180,E1 -9377.905,E2 -9377.905} C_VEL
LIN {X 0,Y 434.915,Z 230.869,A -85,B 0,C 180,E1 -9378.039,E2 -9378.039} C_VEL
LIN {X 0,Y 434.603,Z 226.107,A -85,B 0,C 180,E1 -9379.36,E2 -9379.36} C_VEL
LIN {X 0,Y 433.192,Z 219.31,A -85,B 0,C 180,E1 -9381.41,E2 -9381.41} C_VEL
LIN {X 0,Y 432.351,Z 215.633,A -85,B 0,C 180,E1 -9382.599,E2 -9382.599} C_VEL
LIN {X 0,Y 432.351,Z 215.633,A -85,B 0,C 180,E1 -9385.001,E2 -9385.001} C_VEL
LIN {X 0,Y 432.387,Z 215.628,A -85,B 0,C 180,E1 -9388.123,E2 -9388.123} C_VEL
LIN {X 0,Y 432.326,Z 215.632,A -85,B 0,C 180,E1 -9391.346,E2 -9391.346} C_VEL
LIN {X 0,Y 432.345,Z 215.63,A -85,B 0,C 180,E1 -9394.677,E2 -9394.677} C_VEL
LIN {X 0,Y 432.342,Z 215.632,A -85,B 0,C 180,E1 -9398.149,E2 -9398.149} C_VEL
LIN {X 0,Y 432.338,Z 215.631,A -85,B 0,C 180,E1 -9401.601,E2 -9401.601} C_VEL
LIN {X 0,Y 432.338,Z 215.634,A -85,B 0,C 180,E1 -9404.347,E2 -9404.347} C_VEL
LIN {X 0,Y 432.321,Z 215.632,A -85,B 0,C 180,E1 -9407.016,E2 -9407.016} C_VEL
LIN {X 0,Y 432.336,Z 215.632,A -85,B 0,C 180,E1 -9409.82,E2 -9409.82} C_VEL
LIN {X 0,Y 432.309,Z 215.635,A -85,B 0,C 180,E1 -9413.021,E2 -9413.021} C_VEL
LIN {X 0,Y 432.364,Z 215.632,A -85,B 0,C 180,E1 -9415.996,E2 -9415.996} C_VEL
LIN {X 0,Y 432.351,Z 215.638,A -85,B 0,C 180,E1 -9419.489,E2 -9419.489} C_VEL
LIN {X 0,Y 432.401,Z 215.79,A -85,B 0,C 180,E1 -9420.816,E2 -9420.816} C_VEL
LIN {X 0,Y 434.581,Z 224.667,A -85,B 0,C 180,E1 -9423.075,E2 -9423.075} C_VEL
LIN {X 0,Y 436.105,Z 232.928,A -85,B 0,C 180,E1 -9424.994,E2 -9424.994} C_VEL
LIN {X 0,Y 435.186,Z 245.056,A -85,B 0,C 180,E1 -9427.445,E2 -9427.445} C_VEL
LIN {X 0,Y 433.864,Z 263.188,A -85,B 0,C 180,E1 -9430.942,E2 -9430.942} C_VEL
LIN {X 0,Y 436.922,Z 280.541,A -85,B 0,C 180,E1 -9431.549,E2 -9431.549} C_VEL
LIN {X 0,Y 437.989,Z 291.22,A -85,B 0,C 180,E1 -9431.863,E2 -9431.863} C_VEL
LIN {X 0,Y 436.215,Z 374.335,A -85,B 0,C 180,E1 -9433.653,E2 -9433.653} C_VEL
LIN {X 0,Y 435.72,Z 386.947,A -85,B 0,C 180,E1 -9434.084,E2 -9434.084} C_VEL
LIN {X 0,Y 435.08,Z 399.014,A -85,B 0,C 180,E1 -9434.661,E2 -9434.661} C_VEL
LIN {X 0,Y 434.332,Z 411.675,A -85,B 0,C 180,E1 -9435.474,E2 -9435.474} C_VEL
LIN {X 0,Y 433.689,Z 422.789,A -85,B 0,C 180,E1 -9436.383,E2 -9436.383} C_VEL
LIN {X 0,Y 433.009,Z 433.448,A -85,B 0,C 180,E1 -9437.461,E2 -9437.461} C_VEL
LIN {X 0,Y 432.447,Z 443.688,A -85,B 0,C 180,E1 -9438.753,E2 -9438.753} C_VEL
LIN {X 0,Y 431.93,Z 452.726,A -85,B 0,C 180,E1 -9440.162,E2 -9440.162} C_VEL
LIN {X 0,Y 431.605,Z 459.953,A -85,B 0,C 180,E1 -9441.572,E2 -9441.572} C_VEL
LIN {X 0,Y 431.393,Z 465.751,A -85,B 0,C 180,E1 -9442.981,E2 -9442.981} C_VEL
LIN {X 0,Y 431.264,Z 470.302,A -85,B 0,C 180,E1 -9444.388,E2 -9444.388} C_VEL
LIN {X 0,Y 431.274,Z 472.723,A -85,B 0,C 180,E1 -9445.325,E2 -9445.325} C_VEL
LIN {X 0,Y 431.198,Z 474.643,A -85,B 0,C 180,E1 -9446.261,E2 -9446.261} C_VEL
LIN {X 0,Y 431.28,Z 476.105,A -85,B 0,C 180,E1 -9447.197,E2 -9447.197} C_VEL
LIN {X 0,Y 431.241,Z 477.143,A -85,B 0,C 180,E1 -9448.131,E2 -9448.131} C_VEL
LIN {X 0,Y 431.222,Z 477.756,A -85,B 0,C 180,E1 -9449.065,E2 -9449.065} C_VEL
LIN {X 0,Y 431.238,Z 477.9,A -85,B 0,C 180,E1 -9449.999,E2 -9449.999} C_VEL
LIN {X 0,Y 431.221,Z 477.625,A -85,B 0,C 180,E1 -9450.933,E2 -9450.933} C_VEL
LIN {X 0,Y 431.241,Z 476.938,A -85,B 0,C 180,E1 -9451.867,E2 -9451.867} C_VEL
LIN {X 0,Y 431.305,Z 475.8,A -85,B 0,C 180,E1 -9452.801,E2 -9452.801} C_VEL
LIN {X 0,Y 431.228,Z 473.242,A -85,B 0,C 180,E1 -9454.205,E2 -9454.205} C_VEL
LIN {X 0,Y 431.274,Z 469.613,A -85,B 0,C 180,E1 -9455.61,E2 -9455.61} C_VEL
LIN {X 0,Y 431.396,Z 464.811,A -85,B 0,C 180,E1 -9457.017,E2 -9457.017} C_VEL
LIN {X 0,Y 431.634,Z 458.098,A -85,B 0,C 180,E1 -9458.661,E2 -9458.661} C_VEL
LIN {X 0,Y 431.968,Z 450.892,A -85,B 0,C 180,E1 -9460.072,E2 -9460.072} C_VEL
LIN {X 0,Y 432.546,Z 441.948,A -85,B 0,C 180,E1 -9461.48,E2 -9461.48} C_VEL
LIN {X 0,Y 433.105,Z 432.73,A -85,B 0,C 180,E1 -9462.653,E2 -9462.653} C_VEL
LIN {X 0,Y 433.72,Z 422.325,A -85,B 0,C 180,E1 -9463.719,E2 -9463.719} C_VEL
LIN {X 0,Y 434.475,Z 411.047,A -85,B 0,C 180,E1 -9464.639,E2 -9464.639} C_VEL
LIN {X 0,Y 435.14,Z 399.069,A -85,B 0,C 180,E1 -9465.395,E2 -9465.395} C_VEL
LIN {X 0,Y 435.746,Z 385.733,A -85,B 0,C 180,E1 -9466.003,E2 -9466.003} C_VEL
LIN {X 0,Y 436.282,Z 373.376,A -85,B 0,C 180,E1 -9466.373,E2 -9466.373} C_VEL
LIN {X 0,Y 436.984,Z 288.834,A -85,B 0,C 180,E1 -9467.823,E2 -9467.823} C_VEL
LIN {X 0,Y 433.436,Z 264.574,A -85,B 0,C 180,E1 -9468.433,E2 -9468.433} C_VEL
LIN {X 0,Y 434.511,Z 244.578,A -85,B 0,C 180,E1 -9472.088,E2 -9472.088} C_VEL
LIN {X 0,Y 435.346,Z 231.226,A -85,B 0,C 180,E1 -9474.562,E2 -9474.562} C_VEL
LIN {X 0,Y 433.65,Z 221.781,A -85,B 0,C 180,E1 -9476.446,E2 -9476.446} C_VEL
LIN {X 0,Y 432.446,Z 215.62,A -85,B 0,C 180,E1 -9477.722,E2 -9477.722} C_VEL
LIN {X 0,Y 432.318,Z 215.632,A -85,B 0,C 180,E1 -9481.345,E2 -9481.345} C_VEL
LIN {X 0,Y 432.335,Z 215.62,A -85,B 0,C 180,E1 -9484.676,E2 -9484.676} C_VEL
LIN {X 0,Y 432.324,Z 215.628,A -85,B 0,C 180,E1 -9488.15,E2 -9488.15} C_VEL
LIN {X 0,Y 432.314,Z 215.633,A -85,B 0,C 180,E1 -9491.798,E2 -9491.798} C_VEL
LIN {X 0,Y 432.327,Z 215.628,A -85,B 0,C 180,E1 -9494.346,E2 -9494.346} C_VEL
LIN {X 0,Y 432.3,Z 215.634,A -85,B 0,C 180,E1 -9497.017,E2 -9497.017} C_VEL
LIN {X 0,Y 432.283,Z 215.637,A -85,B 0,C 180,E1 -9499.827,E2 -9499.827} C_VEL
LIN {X 0,Y 432.298,Z 215.631,A -85,B 0,C 180,E1 -9503.021,E2 -9503.021} C_VEL
LIN {X 0,Y 432.35,Z 215.623,A -85,B 0,C 180,E1 -9505.996,E2 -9505.996} C_VEL
LIN {X 0,Y 432.337,Z 215.618,A -85,B 0,C 180,E1 -9509.49,E2 -9509.49} C_VEL
LIN {X 0,Y 432.318,Z 215.622,A -85,B 0,C 180,E1 -9511.872,E2 -9511.872} C_VEL
LIN {X 0,Y 432.34,Z 215.622,A -85,B 0,C 180,E1 -9515.547,E2 -9515.547} C_VEL
LIN {X 0,Y 432.339,Z 215.617,A -85,B 0,C 180,E1 -9519.046,E2 -9519.046} C_VEL
LIN {X 0,Y 432.347,Z 215.626,A -85,B 0,C 180,E1 -9522.01,E2 -9522.01} C_VEL
LIN {X 0,Y 432.355,Z 215.613,A -85,B 0,C 180,E1 -9524.925,E2 -9524.925} C_VEL
LIN {X 0,Y 432.449,Z 215.606,A -85,B 0,C 180,E1 -9527.803,E2 -9527.803} C_VEL
LIN {X 0,Y 432.453,Z 215.612,A -85,B 0,C 180,E1 -9531.59,E2 -9531.59} C_VEL
LIN {X 0,Y 432.537,Z 215.589,A -85,B 0,C 180,E1 -9534.406,E2 -9534.406} C_VEL
LIN {X 0,Y 432.592,Z 215.597,A -85,B 0,C 180,E1 -9538.138,E2 -9538.138} C_VEL
LIN {X 0,Y 432.547,Z 215.593,A -85,B 0,C 180,E1 -9540.931,E2 -9540.931} C_VEL
LIN {X 0,Y 432.557,Z 215.584,A -85,B 0,C 180,E1 -9542.794,E2 -9542.794} C_VEL
LIN {X 0,Y 432.584,Z 215.593,A -85,B 0,C 180,E1 -9545.594,E2 -9545.594} C_VEL
LIN {X 0,Y 432.483,Z 215.603,A -85,B 0,C 180,E1 -9548.41,E2 -9548.41} C_VEL
LIN {X 0,Y 432.451,Z 215.612,A -85,B 0,C 180,E1 -9552.197,E2 -9552.197} C_VEL
LIN {X 0,Y 432.422,Z 215.611,A -85,B 0,C 180,E1 -9556.04,E2 -9556.04} C_VEL
LIN {X 0,Y 432.379,Z 215.622,A -85,B 0,C 180,E1 -9559.486,E2 -9559.486} C_VEL
LIN {X 0,Y 432.312,Z 215.627,A -85,B 0,C 180,E1 -9562.965,E2 -9562.965} C_VEL
LIN {X 0,Y 432.358,Z 215.628,A -85,B 0,C 180,E1 -9566.033,E2 -9566.033} C_VEL
LIN {X 0,Y 432.336,Z 215.625,A -85,B 0,C 180,E1 -9569.188,E2 -9569.188} C_VEL
LIN {X 0,Y 432.317,Z 215.632,A -85,B 0,C 180,E1 -9572.444,E2 -9572.444} C_VEL
LIN {X 0,Y 432.34,Z 215.633,A -85,B 0,C 180,E1 -9575.633,E2 -9575.633} C_VEL
LIN {X 0,Y 432.348,Z 215.625,A -85,B 0,C 180,E1 -9578.718,E2 -9578.718} C_VEL
LIN {X 0,Y 432.33,Z 215.627,A -85,B 0,C 180,E1 -9581.798,E2 -9581.798} C_VEL
LIN {X 0,Y 432.337,Z 215.631,A -85,B 0,C 180,E1 -9584.348,E2 -9584.348} C_VEL
LIN {X 0,Y 432.321,Z 215.633,A -85,B 0,C 180,E1 -9587.016,E2 -9587.016} C_VEL
LIN {X 0,Y 432.334,Z 215.628,A -85,B 0,C 180,E1 -9589.822,E2 -9589.822} C_VEL
LIN {X 0,Y 432.305,Z 215.636,A -85,B 0,C 180,E1 -9593.023,E2 -9593.023} C_VEL
LIN {X 0,Y 432.392,Z 215.628,A -85,B 0,C 180,E1 -9596.479,E2 -9596.479} C_VEL
LIN {X 0,Y 434.067,Z 222.869,A -85,B 0,C 180,E1 -9597.305,E2 -9597.305} C_VEL
LIN {X 0,Y 438.113,Z 244.42,A -85,B 0,C 180,E1 -9597.887,E2 -9597.887} C_VEL
LIN {X 0,Y 437.029,Z 334.889,A -85,B 0,C 180,E1 -9599.416,E2 -9599.416} C_VEL
LIN {X 0,Y 436.673,Z 347.744,A -85,B 0,C 180,E1 -9599.806,E2 -9599.806} C_VEL
LIN {X 0,Y 436.268,Z 359.392,A -85,B 0,C 180,E1 -9600.336,E2 -9600.336} C_VEL
LIN {X 0,Y 435.735,Z 371.221,A -85,B 0,C 180,E1 -9601.063,E2 -9601.063} C_VEL
LIN {X 0,Y 435.022,Z 382.307,A -85,B 0,C 180,E1 -9601.933,E2 -9601.933} C_VEL
LIN {X 0,Y 434.385,Z 391.756,A -85,B 0,C 180,E1 -9602.856,E2 -9602.856} C_VEL
LIN {X 0,Y 433.709,Z 401.667,A -85,B 0,C 180,E1 -9604.056,E2 -9604.056} C_VEL
LIN {X 0,Y 432.995,Z 411.061,A -85,B 0,C 180,E1 -9605.469,E2 -9605.469} C_VEL
LIN {X 0,Y 432.515,Z 418.136,A -85,B 0,C 180,E1 -9606.795,E2 -9606.795} C_VEL
LIN {X 0,Y 432.144,Z 423.55,A -85,B 0,C 180,E1 -9608.036,E2 -9608.036} C_VEL
LIN {X 0,Y 431.744,Z 428.706,A -85,B 0,C 180,E1 -9609.515,E2 -9609.515} C_VEL
LIN {X 0,Y 431.538,Z 432.613,A -85,B 0,C 180,E1 -9610.992,E2 -9610.992} C_VEL
LIN {X 0,Y 431.364,Z 434.592,A -85,B 0,C 180,E1 -9611.969,E2 -9611.969} C_VEL
LIN {X 0,Y 431.246,Z 436.127,A -85,B 0,C 180,E1 -9612.943,E2 -9612.943} C_VEL
LIN {X 0,Y 431.207,Z 437.279,A -85,B 0,C 180,E1 -9614.045,E2 -9614.045} C_VEL
LIN {X 0,Y 430.577,Z 437.824,A -85,B 0,C 180,E1 -9614.822,E2 -9614.822} C_VEL
LIN {X 0,Y 427.705,Z 438.171,A -85,B 0,C 180,E1 -9616.088,E2 -9616.088} C_VEL
LIN {X 0,Y 425.259,Z 437.92,A -85,B 0,C 180,E1 -9617.11,E2 -9617.11} C_VEL
LIN {X 0,Y 424.217,Z 437.387,A -85,B 0,C 180,E1 -9617.896,E2 -9617.896} C_VEL
LIN {X 0,Y 424.139,Z 437.104,A -85,B 0,C 180,E1 -9618.162,E2 -9618.162} C_VEL
LIN {X 0,Y 424.182,Z 435.365,A -85,B 0,C 180,E1 -9619.5,E2 -9619.5} C_VEL
LIN {X 0,Y 424.352,Z 432.49,A -85,B 0,C 180,E1 -9620.949,E2 -9620.949} C_VEL
LIN {X 0,Y 424.567,Z 428.579,A -85,B 0,C 180,E1 -9622.391,E2 -9622.391} C_VEL
LIN {X 0,Y 424.841,Z 423.521,A -85,B 0,C 180,E1 -9623.828,E2 -9623.828} C_VEL
LIN {X 0,Y 425.202,Z 417.148,A -85,B 0,C 180,E1 -9625.261,E2 -9625.261} C_VEL
LIN {X 0,Y 425.663,Z 409.239,A -85,B 0,C 180,E1 -9626.688,E2 -9626.688} C_VEL
LIN {X 0,Y 426.207,Z 401.16,A -85,B 0,C 180,E1 -9627.875,E2 -9627.875} C_VEL
LIN {X 0,Y 426.833,Z 391.277,A -85,B 0,C 180,E1 -9629.058,E2 -9629.058} C_VEL
LIN {X 0,Y 427.539,Z 380.182,A -85,B 0,C 180,E1 -9630.119,E2 -9630.119} C_VEL
LIN {X 0,Y 428.109,Z 369.367,A -85,B 0,C 180,E1 -9630.942,E2 -9630.942} C_VEL
LIN {X 0,Y 428.543,Z 357.367,A -85,B 0,C 180,E1 -9631.646,E2 -9631.646} C_VEL
LIN {X 0,Y 428.982,Z 344.344,A -85,B 0,C 180,E1 -9632.195,E2 -9632.195} C_VEL
LIN {X 0,Y 429.247,Z 331.002,A -85,B 0,C 180,E1 -9632.552,E2 -9632.552} C_VEL
LIN {X 0,Y 430.089,Z 244.175,A -85,B 0,C 180,E1 -9634.007,E2 -9634.007} C_VEL
LIN {X 0,Y 426.329,Z 222.448,A -85,B 0,C 180,E1 -9634.551,E2 -9634.551} C_VEL
LIN {X 0,Y 425.47,Z 216.492,A -85,B 0,C 180,E1 -9635.243,E2 -9635.243} C_VEL
LIN {X 0,Y 425.511,Z 216.484,A -85,B 0,C 180,E1 -9637.69,E2 -9637.69} C_VEL
LIN {X 0,Y 425.354,Z 216.5,A -85,B 0,C 180,E1 -9641.437,E2 -9641.437} C_VEL
LIN {X 0,Y 425.351,Z 216.502,A -85,B 0,C 180,E1 -9644.351,E2 -9644.351} C_VEL
LIN {X 0,Y 425.346,Z 216.501,A -85,B 0,C 180,E1 -9647.303,E2 -9647.303} C_VEL
LIN {X 0,Y 425.302,Z 216.508,A -85,B 0,C 180,E1 -9650.306,E2 -9650.306} C_VEL
LIN {X 0,Y 425.276,Z 216.51,A -85,B 0,C 180,E1 -9653.368,E2 -9653.368} C_VEL
LIN {X 0,Y 425.293,Z 216.51,A -85,B 0,C 180,E1 -9656.5,E2 -9656.5} C_VEL
LIN {X 0,Y 425.287,Z 216.51,A -85,B 0,C 180,E1 -9659.721,E2 -9659.721} C_VEL
LIN {X 0,Y 425.275,Z 216.51,A -85,B 0,C 180,E1 -9663.05,E2 -9663.05} C_VEL
LIN {X 0,Y 425.285,Z 216.511,A -85,B 0,C 180,E1 -9665.928,E2 -9665.928} C_VEL
LIN {X 0,Y 425.251,Z 216.514,A -85,B 0,C 180,E1 -9669.035,E2 -9669.035} C_VEL
LIN {X 0,Y 425.26,Z 216.512,A -85,B 0,C 180,E1 -9672.656,E2 -9672.656} C_VEL
LIN {X 0,Y 425.289,Z 216.509,A -85,B 0,C 180,E1 -9675.284,E2 -9675.284} C_VEL
LIN {X 0,Y 425.25,Z 216.514,A -85,B 0,C 180,E1 -9678.618,E2 -9678.618} C_VEL
LIN {X 0,Y 425.271,Z 216.511,A -85,B 0,C 180,E1 -9682.304,E2 -9682.304} C_VEL
LIN {X 0,Y 425.274,Z 216.511,A -85,B 0,C 180,E1 -9685.814,E2 -9685.814} C_VEL
LIN {X 0,Y 425.291,Z 216.51,A -85,B 0,C 180,E1 -9689.241,E2 -9689.241} C_VEL
LIN {X 0,Y 425.243,Z 216.516,A -85,B 0,C 180,E1 -9692.434,E2 -9692.434} C_VEL
LIN {X 0,Y 425.325,Z 216.504,A -85,B 0,C 180,E1 -9695.6,E2 -9695.6} C_VEL
LIN {X 0,Y 425.331,Z 216.623,A -85,B 0,C 180,E1 -9697.953,E2 -9697.953} C_VEL
LIN {X 0,Y 426.609,Z 224.387,A -85,B 0,C 180,E1 -9699.89,E2 -9699.89} C_VEL
LIN {X 0,Y 426.573,Z 227.808,A -85,B 0,C 180,E1 -9700.704,E2 -9700.704} C_VEL
LIN {X 0,Y 429.981,Z 245.806,A -85,B 0,C 180,E1 -9701.209,E2 -9701.209} C_VEL
LIN {X 0,Y 428.425,Z 335.99,A -85,B 0,C 180,E1 -9703.041,E2 -9703.041} C_VEL
LIN {X 0,Y 428.104,Z 349.008,A -85,B 0,C 180,E1 -9703.488,E2 -9703.488} C_VEL
LIN {X 0,Y 427.773,Z 361.224,A -85,B 0,C 180,E1 -9704.087,E2 -9704.087} C_VEL
LIN {X 0,Y 427.236,Z 373.095,A -85,B 0,C 180,E1 -9704.862,E2 -9704.862} C_VEL
LIN {X 0,Y 426.669,Z 384.739,A -85,B 0,C 180,E1 -9705.829,E2 -9705.829} C_VEL
LIN {X 0,Y 426.162,Z 395.569,A -85,B 0,C 180,E1 -9706.96,E2 -9706.96} C_VEL
LIN {X 0,Y 425.736,Z 404.373,A -85,B 0,C 180,E1 -9708.091,E2 -9708.091} C_VEL
LIN {X 0,Y 425.208,Z 413.492,A -85,B 0,C 180,E1 -9709.524,E2 -9709.524} C_VEL
LIN {X 0,Y 424.889,Z 420.76,A -85,B 0,C 180,E1 -9710.959,E2 -9710.959} C_VEL
LIN {X 0,Y 424.578,Z 426.55,A -85,B 0,C 180,E1 -9712.39,E2 -9712.39} C_VEL
LIN {X 0,Y 424.431,Z 430.93,A -85,B 0,C 180,E1 -9713.765,E2 -9713.765} C_VEL
LIN {X 0,Y 424.291,Z 434.485,A -85,B 0,C 180,E1 -9715.249,E2 -9715.249} C_VEL
LIN {X 0,Y 424.28,Z 436.183,A -85,B 0,C 180,E1 -9716.201,E2 -9716.201} C_VEL
LIN {X 0,Y 424.298,Z 437.44,A -85,B 0,C 180,E1 -9717.151,E2 -9717.151} C_VEL
LIN {X 0,Y 424.2,Z 438.237,A -85,B 0,C 180,E1 -9718.101,E2 -9718.101} C_VEL
LIN {X 0,Y 424.158,Z 438.629,A -85,B 0,C 180,E1 -9719.05,E2 -9719.05} C_VEL
LIN {X 0,Y 424.185,Z 438.612,A -85,B 0,C 180,E1 -9720,E2 -9720} C_VEL
LIN {X 0,Y 424.235,Z 438.139,A -85,B 0,C 180,E1 -9720.949,E2 -9720.949} C_VEL
LIN {X 0,Y 424.302,Z 437.24,A -85,B 0,C 180,E1 -9721.898,E2 -9721.898} C_VEL
LIN {X 0,Y 424.446,Z 435.928,A -85,B 0,C 180,E1 -9722.847,E2 -9722.847} C_VEL
LIN {X 0,Y 424.623,Z 433.108,A -85,B 0,C 180,E1 -9724.271,E2 -9724.271} C_VEL
LIN {X 0,Y 424.703,Z 429.232,A -85,B 0,C 180,E1 -9725.698,E2 -9725.698} C_VEL
LIN {X 0,Y 425.126,Z 424.685,A -85,B 0,C 180,E1 -9726.985,E2 -9726.985} C_VEL
LIN {X 0,Y 425.568,Z 417.775,A -85,B 0,C 180,E1 -9728.547,E2 -9728.547} C_VEL
LIN {X 0,Y 426.156,Z 409.75,A -85,B 0,C 180,E1 -9729.972,E2 -9729.972} C_VEL
LIN {X 0,Y 426.65,Z 401.569,A -85,B 0,C 180,E1 -9731.16,E2 -9731.16} C_VEL
LIN {X 0,Y 427.273,Z 391.612,A -85,B 0,C 180,E1 -9732.347,E2 -9732.347} C_VEL
LIN {X 0,Y 428.105,Z 380.356,A -85,B 0,C 180,E1 -9733.408,E2 -9733.408} C_VEL
LIN {X 0,Y 428.738,Z 368.097,A -85,B 0,C 180,E1 -9734.329,E2 -9734.329} C_VEL
LIN {X 0,Y 429.366,Z 355.465,A -85,B 0,C 180,E1 -9735.04,E2 -9735.04} C_VEL
LIN {X 0,Y 429.764,Z 342.093,A -85,B 0,C 180,E1 -9735.593,E2 -9735.593} C_VEL
LIN {X 0,Y 430.124,Z 327.094,A -85,B 0,C 180,E1 -9735.975,E2 -9735.975} C_VEL
LIN {X 0,Y 432.159,Z 251.714,A -85,B 0,C 180,E1 -9737.655,E2 -9737.655} C_VEL
LIN {X 0,Y 432.098,Z 246.531,A -85,B 0,C 180,E1 -9737.789,E2 -9737.789} C_VEL
LIN {X 0,Y 429.163,Z 234.922,A -85,B 0,C 180,E1 -9738.281,E2 -9738.281} C_VEL
LIN {X 0,Y 428.103,Z 231.473,A -85,B 0,C 180,E1 -9738.46,E2 -9738.46} C_VEL
LIN {X 0,Y 427.377,Z 225.531,A -85,B 0,C 180,E1 -9740.202,E2 -9740.202} C_VEL
LIN {X 0,Y 425.29,Z 216.512,A -85,B 0,C 180,E1 -9743.108,E2 -9743.108} C_VEL
LIN {X 0,Y 425.296,Z 216.511,A -85,B 0,C 180,E1 -9745.445,E2 -9745.445} C_VEL
LIN {X 0,Y 425.354,Z 216.503,A -85,B 0,C 180,E1 -9747.557,E2 -9747.557} C_VEL
LIN {X 0,Y 425.293,Z 216.509,A -85,B 0,C 180,E1 -9750.816,E2 -9750.816} C_VEL
LIN {X 0,Y 425.317,Z 216.509,A -85,B 0,C 180,E1 -9754.287,E2 -9754.287} C_VEL
LIN {X 0,Y 425.284,Z 216.51,A -85,B 0,C 180,E1 -9757.694,E2 -9757.694} C_VEL
LIN {X 0,Y 425.285,Z 216.509,A -85,B 0,C 180,E1 -9760.52,E2 -9760.52} C_VEL
LIN {X 0,Y 425.262,Z 216.513,A -85,B 0,C 180,E1 -9763.35,E2 -9763.35} C_VEL
LIN {X 0,Y 425.26,Z 216.512,A -85,B 0,C 180,E1 -9766.649,E2 -9766.649} C_VEL
LIN {X 0,Y 425.288,Z 216.51,A -85,B 0,C 180,E1 -9769.872,E2 -9769.872} C_VEL
LIN {X 0,Y 425.28,Z 216.512,A -85,B 0,C 180,E1 -9772.488,E2 -9772.488} C_VEL
LIN {X 0,Y 425.312,Z 216.509,A -85,B 0,C 180,E1 -9775.817,E2 -9775.817} C_VEL
LIN {X 0,Y 425.295,Z 216.517,A -85,B 0,C 180,E1 -9779.238,E2 -9779.238} C_VEL
LIN {X 0,Y 425.348,Z 216.714,A -85,B 0,C 180,E1 -9780.284,E2 -9780.284} C_VEL
LIN {X 0,Y 427.707,Z 226.222,A -85,B 0,C 180,E1 -9782.809,E2 -9782.809} C_VEL
LIN {X 0,Y 429.314,Z 234.535,A -85,B 0,C 180,E1 -9784.809,E2 -9784.809} C_VEL
LIN {X 0,Y 428.555,Z 244.209,A -85,B 0,C 180,E1 -9786.821,E2 -9786.821} C_VEL
LIN {X 0,Y 427.056,Z 262.817,A -85,B 0,C 180,E1 -9790.502,E2 -9790.502} C_VEL
LIN {X 0,Y 430.047,Z 279.026,A -85,B 0,C 180,E1 -9791.103,E2 -9791.103} C_VEL
LIN {X 0,Y 431.463,Z 291.442,A -85,B 0,C 180,E1 -9791.496,E2 -9791.496} C_VEL
LIN {X 0,Y 429.489,Z 374.881,A -85,B 0,C 180,E1 -9793.359,E2 -9793.359} C_VEL
LIN {X 0,Y 428.945,Z 387.849,A -85,B 0,C 180,E1 -9793.826,E2 -9793.826} C_VEL
LIN {X 0,Y 428.266,Z 399.476,A -85,B 0,C 180,E1 -9794.411,E2 -9794.411} C_VEL
LIN {X 0,Y 427.478,Z 411.913,A -85,B 0,C 180,E1 -9795.236,E2 -9795.236} C_VEL
LIN {X 0,Y 426.735,Z 423.698,A -85,B 0,C 180,E1 -9796.232,E2 -9796.232} C_VEL
LIN {X 0,Y 426.009,Z 434.441,A -85,B 0,C 180,E1 -9797.373,E2 -9797.373} C_VEL
LIN {X 0,Y 425.476,Z 443.611,A -85,B 0,C 180,E1 -9798.566,E2 -9798.566} C_VEL
LIN {X 0,Y 424.941,Z 451.209,A -85,B 0,C 180,E1 -9799.758,E2 -9799.758} C_VEL
LIN {X 0,Y 424.605,Z 458.71,A -85,B 0,C 180,E1 -9801.192,E2 -9801.192} C_VEL
LIN {X 0,Y 424.374,Z 463.785,A -85,B 0,C 180,E1 -9802.386,E2 -9802.386} C_VEL
LIN {X 0,Y 424.224,Z 468.413,A -85,B 0,C 180,E1 -9803.724,E2 -9803.724} C_VEL
LIN {X 0,Y 424.201,Z 472.476,A -85,B 0,C 180,E1 -9805.247,E2 -9805.247} C_VEL
LIN {X 0,Y 424.109,Z 474.367,A -85,B 0,C 180,E1 -9806.198,E2 -9806.198} C_VEL
LIN {X 0,Y 424.176,Z 475.816,A -85,B 0,C 180,E1 -9807.15,E2 -9807.15} C_VEL
LIN {X 0,Y 424.165,Z 476.842,A -85,B 0,C 180,E1 -9808.1,E2 -9808.1} C_VEL
LIN {X 0,Y 424.138,Z 477.426,A -85,B 0,C 180,E1 -9809.05,E2 -9809.05} C_VEL
LIN {X 0,Y 424.151,Z 477.551,A -85,B 0,C 180,E1 -9809.999,E2 -9809.999} C_VEL
LIN {X 0,Y 424.138,Z 477.259,A -85,B 0,C 180,E1 -9810.948,E2 -9810.948} C_VEL
LIN {X 0,Y 424.166,Z 476.553,A -85,B 0,C 180,E1 -9811.898,E2 -9811.898} C_VEL
LIN {X 0,Y 424.215,Z 475.375,A -85,B 0,C 180,E1 -9812.848,E2 -9812.848} C_VEL
LIN {X 0,Y 424.15,Z 472.769,A -85,B 0,C 180,E1 -9814.275,E2 -9814.275} C_VEL
LIN {X 0,Y 424.177,Z 469.084,A -85,B 0,C 180,E1 -9815.704,E2 -9815.704} C_VEL
LIN {X 0,Y 424.378,Z 462.79,A -85,B 0,C 180,E1 -9817.612,E2 -9817.612} C_VEL
LIN {X 0,Y 424.686,Z 455.715,A -85,B 0,C 180,E1 -9819.284,E2 -9819.284} C_VEL
LIN {X 0,Y 425.129,Z 448.058,A -85,B 0,C 180,E1 -9820.717,E2 -9820.717} C_VEL
LIN {X 0,Y 425.802,Z 438.429,A -85,B 0,C 180,E1 -9822.147,E2 -9822.147} C_VEL
LIN {X 0,Y 426.395,Z 428.486,A -85,B 0,C 180,E1 -9823.34,E2 -9823.34} C_VEL
LIN {X 0,Y 427.229,Z 417.233,A -85,B 0,C 180,E1 -9824.406,E2 -9824.406} C_VEL
LIN {X 0,Y 427.949,Z 406.199,A -85,B 0,C 180,E1 -9825.233,E2 -9825.233} C_VEL
LIN {X 0,Y 428.598,Z 395.054,A -85,B 0,C 180,E1 -9825.88,E2 -9825.88} C_VEL
LIN {X 0,Y 429.17,Z 382.545,A -85,B 0,C 180,E1 -9826.407,E2 -9826.407} C_VEL
LIN {X 0,Y 429.604,Z 369.435,A -85,B 0,C 180,E1 -9826.757,E2 -9826.757} C_VEL
LIN {X 0,Y 430.403,Z 290.341,A -85,B 0,C 180,E1 -9828.119,E2 -9828.119} C_VEL
LIN {X 0,Y 426.466,Z 263.71,A -85,B 0,C 180,E1 -9828.799,E2 -9828.799} C_VEL
LIN {X 0,Y 427.518,Z 245.353,A -85,B 0,C 180,E1 -9832.215,E2 -9832.215} C_VEL
LIN {X 0,Y 428.343,Z 232.015,A -85,B 0,C 180,E1 -9834.732,E2 -9834.732} C_VEL
LIN {X 0,Y 426.054,Z 219.777,A -85,B 0,C 180,E1 -9837.221,E2 -9837.221} C_VEL
LIN {X 0,Y 425.392,Z 216.499,A -85,B 0,C 180,E1 -9837.954,E2 -9837.954} C_VEL
LIN {X 0,Y 425.284,Z 216.508,A -85,B 0,C 180,E1 -9840.815,E2 -9840.815} C_VEL
LIN {X 0,Y 425.307,Z 216.489,A -85,B 0,C 180,E1 -9844.287,E2 -9844.287} C_VEL
LIN {X 0,Y 425.27,Z 216.512,A -85,B 0,C 180,E1 -9847.694,E2 -9847.694} C_VEL
LIN {X 0,Y 425.241,Z 216.513,A -85,B 0,C 180,E1 -9850.514,E2 -9850.514} C_VEL
LIN {X 0,Y 425.249,Z 216.508,A -85,B 0,C 180,E1 -9853.35,E2 -9853.35} C_VEL
LIN {X 0,Y 425.251,Z 216.512,A -85,B 0,C 180,E1 -9856.043,E2 -9856.043} C_VEL
LIN {X 0,Y 425.244,Z 216.501,A -85,B 0,C 180,E1 -9858.618,E2 -9858.618} C_VEL
LIN {X 0,Y 425.273,Z 216.511,A -85,B 0,C 180,E1 -9861.099,E2 -9861.099} C_VEL
LIN {X 0,Y 425.29,Z 216.493,A -85,B 0,C 180,E1 -9864.663,E2 -9864.663} C_VEL
LIN {X 0,Y 425.255,Z 216.507,A -85,B 0,C 180,E1 -9868.072,E2 -9868.072} C_VEL
LIN {X 0,Y 425.295,Z 216.495,A -85,B 0,C 180,E1 -9871.365,E2 -9871.365} C_VEL
LIN {X 0,Y 425.249,Z 216.51,A -85,B 0,C 180,E1 -9874.552,E2 -9874.552} C_VEL
LIN {X 0,Y 425.282,Z 216.487,A -85,B 0,C 180,E1 -9877.729,E2 -9877.729} C_VEL
LIN {X 0,Y 425.351,Z 216.497,A -85,B 0,C 180,E1 -9880.704,E2 -9880.704} C_VEL
LIN {X 0,Y 425.376,Z 216.49,A -85,B 0,C 180,E1 -9883.688,E2 -9883.688} C_VEL
LIN {X 0,Y 425.402,Z 216.483,A -85,B 0,C 180,E1 -9887.598,E2 -9887.598} C_VEL
LIN {X 0,Y 425.398,Z 216.491,A -85,B 0,C 180,E1 -9891.449,E2 -9891.449} C_VEL
LIN {X 0,Y 425.495,Z 216.466,A -85,B 0,C 180,E1 -9894.313,E2 -9894.313} C_VEL
LIN {X 0,Y 425.561,Z 216.473,A -85,B 0,C 180,E1 -9898.107,E2 -9898.107} C_VEL
LIN {X 0,Y 425.509,Z 216.469,A -85,B 0,C 180,E1 -9900.947,E2 -9900.947} C_VEL
LIN {X 0,Y 425.512,Z 216.461,A -85,B 0,C 180,E1 -9902.84,E2 -9902.84} C_VEL
LIN {X 0,Y 425.54,Z 216.471,A -85,B 0,C 180,E1 -9905.687,E2 -9905.687} C_VEL
LIN {X 0,Y 425.434,Z 216.48,A -85,B 0,C 180,E1 -9908.551,E2 -9908.551} C_VEL
LIN {X 0,Y 425.404,Z 216.49,A -85,B 0,C 180,E1 -9912.402,E2 -9912.402} C_VEL
LIN {X 0,Y 425.38,Z 216.485,A -85,B 0,C 180,E1 -9916.312,E2 -9916.312} C_VEL
LIN {X 0,Y 425.321,Z 216.503,A -85,B 0,C 180,E1 -9919.636,E2 -9919.636} C_VEL
LIN {X 0,Y 425.3,Z 216.499,A -85,B 0,C 180,E1 -9923.366,E2 -9923.366} C_VEL
LIN {X 0,Y 425.341,Z 216.501,A -85,B 0,C 180,E1 -9926.845,E2 -9926.845} C_VEL
LIN {X 0,Y 425.284,Z 216.504,A -85,B 0,C 180,E1 -9929.72,E2 -9929.72} C_VEL
LIN {X 0,Y 425.277,Z 216.512,A -85,B 0,C 180,E1 -9933.049,E2 -9933.049} C_VEL
LIN {X 0,Y 425.279,Z 216.511,A -85,B 0,C 180,E1 -9935.93,E2 -9935.93} C_VEL
LIN {X 0,Y 425.299,Z 216.506,A -85,B 0,C 180,E1 -9939.046,E2 -9939.046} C_VEL
LIN {X 0,Y 425.274,Z 216.508,A -85,B 0,C 180,E1 -9942.654,E2 -9942.654} C_VEL
LIN {X 0,Y 425.265,Z 216.51,A -85,B 0,C 180,E1 -9946.046,E2 -9946.046} C_VEL
LIN {X 0,Y 425.272,Z 216.512,A -85,B 0,C 180,E1 -9948.623,E2 -9948.623} C_VEL
LIN {X 0,Y 425.308,Z 216.507,A -85,B 0,C 180,E1 -9951.104,E2 -9951.104} C_VEL
LIN {X 0,Y 425.301,Z 216.51,A -85,B 0,C 180,E1 -9954.666,E2 -9954.666} C_VEL
LIN {X 0,Y 425.356,Z 216.562,A -85,B 0,C 180,E1 -9956.193,E2 -9956.193} C_VEL
LIN {X 0,Y 427.136,Z 223.186,A -85,B 0,C 180,E1 -9956.942,E2 -9956.942} C_VEL
LIN {X 0,Y 430.202,Z 237.988,A -85,B 0,C 180,E1 -9957.369,E2 -9957.369} C_VEL
LIN {X 0,Y 431.506,Z 246.259,A -85,B 0,C 180,E1 -9957.582,E2 -9957.582} C_VEL
LIN {X 0,Y 430.337,Z 335.267,A -85,B 0,C 180,E1 -9959.11,E2 -9959.11} C_VEL
LIN {X 0,Y 429.949,Z 348.515,A -85,B 0,C 180,E1 -9959.521,E2 -9959.521} C_VEL
LIN {X 0,Y 429.452,Z 361.661,A -85,B 0,C 180,E1 -9960.153,E2 -9960.153} C_VEL
LIN {X 0,Y 428.809,Z 373.974,A -85,B 0,C 180,E1 -9960.953,E2 -9960.953} C_VEL
LIN {X 0,Y 427.976,Z 385.824,A -85,B 0,C 180,E1 -9961.963,E2 -9961.963} C_VEL
LIN {X 0,Y 427.199,Z 396.424,A -85,B 0,C 180,E1 -9963.103,E2 -9963.103} C_VEL
LIN {X 0,Y 426.539,Z 405.843,A -85,B 0,C 180,E1 -9964.374,E2 -9964.374} C_VEL
LIN {X 0,Y 425.794,Z 414.885,A -85,B 0,C 180,E1 -9965.89,E2 -9965.89} C_VEL
LIN {X 0,Y 425.264,Z 421.993,A -85,B 0,C 180,E1 -9967.405,E2 -9967.405} C_VEL
LIN {X 0,Y 424.768,Z 428.401,A -85,B 0,C 180,E1 -9969.163,E2 -9969.163} C_VEL
LIN {X 0,Y 424.502,Z 432.522,A -85,B 0,C 180,E1 -9970.681,E2 -9970.681} C_VEL
LIN {X 0,Y 424.336,Z 434.539,A -85,B 0,C 180,E1 -9971.659,E2 -9971.659} C_VEL
LIN {X 0,Y 424.184,Z 436.152,A -85,B 0,C 180,E1 -9972.65,E2 -9972.65} C_VEL
LIN {X 0,Y 424.12,Z 437.63,A -85,B 0,C 180,E1 -9974.028,E2 -9974.028} C_VEL
LIN {X 0,Y 424.035,Z 438.33,A -85,B 0,C 180,E1 -9975.606,E2 -9975.606} C_VEL
LIN {X 0,Y 424.079,Z 438.227,A -85,B 0,C 180,E1 -9976.586,E2 -9976.586} C_VEL
LIN {X 0,Y 424.139,Z 437.104,A -85,B 0,C 180,E1 -9978.162,E2 -9978.162} C_VEL
LIN {X 0,Y 423.502,Z 436.226,A -85,B 0,C 180,E1 -9978.946,E2 -9978.946} C_VEL
LIN {X 0,Y 420.724,Z 434.264,A -85,B 0,C 180,E1 -9980.211,E2 -9980.211} C_VEL
LIN {X 0,Y 418.414,Z 432.201,A -85,B 0,C 180,E1 -9981.215,E2 -9981.215} C_VEL
LIN {X 0,Y 417.487,Z 430.282,A -85,B 0,C 180,E1 -9981.976,E2 -9981.976} C_VEL
LIN {X 0,Y 417.447,Z 429.556,A -85,B 0,C 180,E1 -9982.23,E2 -9982.23} C_VEL
LIN {X 0,Y 417.761,Z 424.574,A -85,B 0,C 180,E1 -9983.723,E2 -9983.723} C_VEL
LIN {X 0,Y 418.104,Z 418.428,A -85,B 0,C 180,E1 -9985.18,E2 -9985.18} C_VEL
LIN {X 0,Y 418.554,Z 410.727,A -85,B 0,C 180,E1 -9986.632,E2 -9986.632} C_VEL
LIN {X 0,Y 419.24,Z 401.137,A -85,B 0,C 180,E1 -9988.08,E2 -9988.08} C_VEL
LIN {X 0,Y 419.896,Z 391.145,A -85,B 0,C 180,E1 -9989.282,E2 -9989.282} C_VEL
LIN {X 0,Y 420.639,Z 379.943,A -85,B 0,C 180,E1 -9990.36,E2 -9990.36} C_VEL
LIN {X 0,Y 421.246,Z 368.958,A -85,B 0,C 180,E1 -9991.196,E2 -9991.196} C_VEL
LIN {X 0,Y 421.701,Z 356.673,A -85,B 0,C 180,E1 -9991.911,E2 -9991.911} C_VEL
LIN {X 0,Y 422.172,Z 343.47,A -85,B 0,C 180,E1 -9992.461,E2 -9992.461} C_VEL
LIN {X 0,Y 422.381,Z 330.001,A -85,B 0,C 180,E1 -9992.807,E2 -9992.807} C_VEL
LIN {X 0,Y 423.324,Z 245.511,A -85,B 0,C 180,E1 -9994.239,E2 -9994.239} C_VEL
LIN {X 0,Y 419.396,Z 222.704,A -85,B 0,C 180,E1 -9994.807,E2 -9994.807} C_VEL
LIN {X 0,Y 418.482,Z 217.363,A -85,B 0,C 180,E1 -9995.422,E2 -9995.422} C_VEL
LIN {X 0,Y 418.473,Z 217.36,A -85,B 0,C 180,E1 -9997.744,E2 -9997.744} C_VEL
LIN {X 0,Y 418.319,Z 217.376,A -85,B 0,C 180,E1 -10001.632,E2 -10001.632} C_VEL
LIN {X 0,Y 418.306,Z 217.38,A -85,B 0,C 180,E1 -10004.598,E2 -10004.598} C_VEL
LIN {X 0,Y 418.292,Z 217.38,A -85,B 0,C 180,E1 -10007.605,E2 -10007.605} C_VEL
LIN {X 0,Y 418.257,Z 217.387,A -85,B 0,C 180,E1 -10010.664,E2 -10010.664} C_VEL
LIN {X 0,Y 418.262,Z 217.385,A -85,B 0,C 180,E1 -10013.784,E2 -10013.784} C_VEL
LIN {X 0,Y 418.215,Z 217.389,A -85,B 0,C 180,E1 -10017.043,E2 -10017.043} C_VEL
LIN {X 0,Y 418.246,Z 217.389,A -85,B 0,C 180,E1 -10020.273,E2 -10020.273} C_VEL
LIN {X 0,Y 418.239,Z 217.388,A -85,B 0,C 180,E1 -10023.679,E2 -10023.679} C_VEL
LIN {X 0,Y 418.24,Z 217.388,A -85,B 0,C 180,E1 -10027.225,E2 -10027.225} C_VEL
LIN {X 0,Y 418.212,Z 217.391,A -85,B 0,C 180,E1 -10030.95,E2 -10030.95} C_VEL
LIN {X 0,Y 418.207,Z 217.393,A -85,B 0,C 180,E1 -10033.728,E2 -10033.728} C_VEL
LIN {X 0,Y 418.203,Z 217.391,A -85,B 0,C 180,E1 -10036.447,E2 -10036.447} C_VEL
LIN {X 0,Y 418.211,Z 217.391,A -85,B 0,C 180,E1 -10039.133,E2 -10039.133} C_VEL
LIN {X 0,Y 418.233,Z 217.389,A -85,B 0,C 180,E1 -10042.775,E2 -10042.775} C_VEL
LIN {X 0,Y 418.225,Z 217.389,A -85,B 0,C 180,E1 -10046.32,E2 -10046.32} C_VEL
LIN {X 0,Y 418.239,Z 217.387,A -85,B 0,C 180,E1 -10049.727,E2 -10049.727} C_VEL
LIN {X 0,Y 418.206,Z 217.392,A -85,B 0,C 180,E1 -10053.016,E2 -10053.016} C_VEL
LIN {X 0,Y 418.262,Z 217.385,A -85,B 0,C 180,E1 -10056.217,E2 -10056.217} C_VEL
LIN {X 0,Y 418.281,Z 217.543,A -85,B 0,C 180,E1 -10057.821,E2 -10057.821} C_VEL
LIN {X 0,Y 419.577,Z 225.072,A -85,B 0,C 180,E1 -10059.723,E2 -10059.723} C_VEL
LIN {X 0,Y 419.604,Z 228.126,A -85,B 0,C 180,E1 -10060.462,E2 -10060.462} C_VEL
LIN {X 0,Y 423.091,Z 247.305,A -85,B 0,C 180,E1 -10061.002,E2 -10061.002} C_VEL
LIN {X 0,Y 421.495,Z 335.968,A -85,B 0,C 180,E1 -10062.847,E2 -10062.847} C_VEL
LIN {X 0,Y 421.128,Z 349.773,A -85,B 0,C 180,E1 -10063.331,E2 -10063.331} C_VEL
LIN {X 0,Y 420.791,Z 361.842,A -85,B 0,C 180,E1 -10063.941,E2 -10063.941} C_VEL
LIN {X 0,Y 420.233,Z 373.64,A -85,B 0,C 180,E1 -10064.728,E2 -10064.728} C_VEL
LIN {X 0,Y 419.653,Z 385.116,A -85,B 0,C 180,E1 -10065.698,E2 -10065.698} C_VEL
LIN {X 0,Y 419.158,Z 395.697,A -85,B 0,C 180,E1 -10066.82,E2 -10066.82} C_VEL
LIN {X 0,Y 418.632,Z 405.672,A -85,B 0,C 180,E1 -10068.132,E2 -10068.132} C_VEL
LIN {X 0,Y 418.164,Z 413.24,A -85,B 0,C 180,E1 -10069.346,E2 -10069.346} C_VEL
LIN {X 0,Y 417.85,Z 420.665,A -85,B 0,C 180,E1 -10070.805,E2 -10070.805} C_VEL
LIN {X 0,Y 417.536,Z 426.549,A -85,B 0,C 180,E1 -10072.261,E2 -10072.261} C_VEL
LIN {X 0,Y 417.337,Z 431.383,A -85,B 0,C 180,E1 -10073.796,E2 -10073.796} C_VEL
LIN {X 0,Y 417.228,Z 434.645,A -85,B 0,C 180,E1 -10075.168,E2 -10075.168} C_VEL
LIN {X 0,Y 417.184,Z 436.379,A -85,B 0,C 180,E1 -10076.136,E2 -10076.136} C_VEL
LIN {X 0,Y 417.23,Z 437.69,A -85,B 0,C 180,E1 -10077.103,E2 -10077.103} C_VEL
LIN {X 0,Y 417.127,Z 438.533,A -85,B 0,C 180,E1 -10078.069,E2 -10078.069} C_VEL
LIN {X 0,Y 417.077,Z 438.957,A -85,B 0,C 180,E1 -10079.034,E2 -10079.034} C_VEL
LIN {X 0,Y 417.099,Z 438.974,A -85,B 0,C 180,E1 -10080,E2 -10080} C_VEL
LIN {X 0,Y 417.151,Z 438.559,A -85,B 0,C 180,E1 -10080.965,E2 -10080.965} C_VEL
LIN {X 0,Y 417.225,Z 437.687,A -85,B 0,C 180,E1 -10081.93,E2 -10081.93} C_VEL
LIN {X 0,Y 417.377,Z 436.402,A -85,B 0,C 180,E1 -10082.895,E2 -10082.895} C_VEL
LIN {X 0,Y 417.58,Z 433.64,A -85,B 0,C 180,E1 -10084.343,E2 -10084.343} C_VEL
LIN {X 0,Y 417.661,Z 429.827,A -85,B 0,C 180,E1 -10085.794,E2 -10085.794} C_VEL
LIN {X 0,Y 418.092,Z 425.592,A -85,B 0,C 180,E1 -10087.037,E2 -10087.037} C_VEL
LIN {X 0,Y 418.599,Z 418.514,A -85,B 0,C 180,E1 -10088.691,E2 -10088.691} C_VEL
LIN {X 0,Y 419.218,Z 410.585,A -85,B 0,C 180,E1 -10090.138,E2 -10090.138} C_VEL
LIN {X 0,Y 419.748,Z 402.507,A -85,B 0,C 180,E1 -10091.346,E2 -10091.346} C_VEL
LIN {X 0,Y 420.442,Z 392.666,A -85,B 0,C 180,E1 -10092.551,E2 -10092.551} C_VEL
LIN {X 0,Y 421.299,Z 381.63,A -85,B 0,C 180,E1 -10093.629,E2 -10093.629} C_VEL
LIN {X 0,Y 421.992,Z 369.567,A -85,B 0,C 180,E1 -10094.567,E2 -10094.567} C_VEL
LIN {X 0,Y 422.625,Z 357.492,A -85,B 0,C 180,E1 -10095.286,E2 -10095.286} C_VEL
LIN {X 0,Y 423.087,Z 343.995,A -85,B 0,C 180,E1 -10095.876,E2 -10095.876} C_VEL
LIN {X 0,Y 423.455,Z 330.258,A -85,B 0,C 180,E1 -10096.264,E2 -10096.264} C_VEL
LIN {X 0,Y 425.732,Z 254.214,A -85,B 0,C 180,E1 -10098.009,E2 -10098.009} C_VEL
LIN {X 0,Y 425.71,Z 247.765,A -85,B 0,C 180,E1 -10098.179,E2 -10098.179} C_VEL
LIN {X 0,Y 423.005,Z 237.135,A -85,B 0,C 180,E1 -10098.654,E2 -10098.654} C_VEL
LIN {X 0,Y 421.253,Z 232.008,A -85,B 0,C 180,E1 -10098.942,E2 -10098.942} C_VEL
LIN {X 0,Y 420.412,Z 226.62,A -85,B 0,C 180,E1 -10100.583,E2 -10100.583} C_VEL
LIN {X 0,Y 418.269,Z 217.387,A -85,B 0,C 180,E1 -10103.716,E2 -10103.716} C_VEL
LIN {X 0,Y 418.316,Z 217.38,A -85,B 0,C 180,E1 -10107.07,E2 -10107.07} C_VEL
LIN {X 0,Y 418.25,Z 217.389,A -85,B 0,C 180,E1 -10110.272,E2 -10110.272} C_VEL
LIN {X 0,Y 418.254,Z 217.385,A -85,B 0,C 180,E1 -10113.677,E2 -10113.677} C_VEL
LIN {X 0,Y 418.245,Z 217.387,A -85,B 0,C 180,E1 -10117.224,E2 -10117.224} C_VEL
LIN {X 0,Y 418.254,Z 217.384,A -85,B 0,C 180,E1 -10119.682,E2 -10119.682} C_VEL
LIN {X 0,Y 418.234,Z 217.388,A -85,B 0,C 180,E1 -10122.321,E2 -10122.321} C_VEL
LIN {X 0,Y 418.24,Z 217.386,A -85,B 0,C 180,E1 -10125.108,E2 -10125.108} C_VEL
LIN {X 0,Y 418.239,Z 217.39,A -85,B 0,C 180,E1 -10127.765,E2 -10127.765} C_VEL
LIN {X 0,Y 418.246,Z 217.386,A -85,B 0,C 180,E1 -10130.621,E2 -10130.621} C_VEL
LIN {X 0,Y 418.247,Z 217.39,A -85,B 0,C 180,E1 -10133.975,E2 -10133.975} C_VEL
LIN {X 0,Y 418.262,Z 217.389,A -85,B 0,C 180,E1 -10137.155,E2 -10137.155} C_VEL
LIN {X 0,Y 418.3,Z 217.526,A -85,B 0,C 180,E1 -10139.671,E2 -10139.671} C_VEL
LIN {X 0,Y 420.496,Z 226.125,A -85,B 0,C 180,E1 -10142.096,E2 -10142.096} C_VEL
LIN {X 0,Y 422.343,Z 235.104,A -85,B 0,C 180,E1 -10144.363,E2 -10144.363} C_VEL
LIN {X 0,Y 422.463,Z 238.644,A -85,B 0,C 180,E1 -10145.161,E2 -10145.161} C_VEL
LIN {X 0,Y 420.993,Z 253.231,A -85,B 0,C 180,E1 -10148.195,E2 -10148.195} C_VEL
LIN {X 0,Y 420.269,Z 262.246,A -85,B 0,C 180,E1 -10150.016,E2 -10150.016} C_VEL
LIN {X 0,Y 423.589,Z 279.807,A -85,B 0,C 180,E1 -10150.712,E2 -10150.712} C_VEL
LIN {X 0,Y 424.973,Z 292.57,A -85,B 0,C 180,E1 -10151.13,E2 -10151.13} C_VEL
LIN {X 0,Y 422.885,Z 373.743,A -85,B 0,C 180,E1 -10152.998,E2 -10152.998} C_VEL
LIN {X 0,Y 422.305,Z 386.112,A -85,B 0,C 180,E1 -10153.44,E2 -10153.44} C_VEL
LIN {X 0,Y 421.566,Z 398.066,A -85,B 0,C 180,E1 -10154.033,E2 -10154.033} C_VEL
LIN {X 0,Y 420.78,Z 410.679,A -85,B 0,C 180,E1 -10154.871,E2 -10154.871} C_VEL
LIN {X 0,Y 419.978,Z 422.096,A -85,B 0,C 180,E1 -10155.833,E2 -10155.833} C_VEL
LIN {X 0,Y 419.166,Z 432.594,A -85,B 0,C 180,E1 -10156.93,E2 -10156.93} C_VEL
LIN {X 0,Y 418.641,Z 441.901,A -85,B 0,C 180,E1 -10158.131,E2 -10158.131} C_VEL
LIN {X 0,Y 417.917,Z 451.14,A -85,B 0,C 180,E1 -10159.584,E2 -10159.584} C_VEL
LIN {X 0,Y 417.545,Z 458.565,A -85,B 0,C 180,E1 -10161.042,E2 -10161.042} C_VEL
LIN {X 0,Y 417.255,Z 465.359,A -85,B 0,C 180,E1 -10162.742,E2 -10162.742} C_VEL
LIN {X 0,Y 417.087,Z 469.851,A -85,B 0,C 180,E1 -10164.196,E2 -10164.196} C_VEL
LIN {X 0,Y 417.106,Z 472.238,A -85,B 0,C 180,E1 -10165.166,E2 -10165.166} C_VEL
LIN {X 0,Y 417.023,Z 474.101,A -85,B 0,C 180,E1 -10166.134,E2 -10166.134} C_VEL
LIN {X 0,Y 417.071,Z 475.534,A -85,B 0,C 180,E1 -10167.101,E2 -10167.101} C_VEL
LIN {X 0,Y 417.091,Z 476.547,A -85,B 0,C 180,E1 -10168.068,E2 -10168.068} C_VEL
LIN {X 0,Y 417.058,Z 477.092,A -85,B 0,C 180,E1 -10169.033,E2 -10169.033} C_VEL
LIN {X 0,Y 417.067,Z 477.199,A -85,B 0,C 180,E1 -10169.999,E2 -10169.999} C_VEL
LIN {X 0,Y 417.058,Z 476.887,A -85,B 0,C 180,E1 -10170.964,E2 -10170.964} C_VEL
LIN {X 0,Y 417.093,Z 476.15,A -85,B 0,C 180,E1 -10171.93,E2 -10171.93} C_VEL
LIN {X 0,Y 417.128,Z 474.931,A -85,B 0,C 180,E1 -10172.896,E2 -10172.896} C_VEL
LIN {X 0,Y 417.076,Z 472.273,A -85,B 0,C 180,E1 -10174.348,E2 -10174.348} C_VEL
LIN {X 0,Y 417.133,Z 467.359,A -85,B 0,C 180,E1 -10176.251,E2 -10176.251} C_VEL
LIN {X 0,Y 417.323,Z 462.608,A -85,B 0,C 180,E1 -10177.742,E2 -10177.742} C_VEL
LIN {X 0,Y 417.651,Z 455.58,A -85,B 0,C 180,E1 -10179.442,E2 -10179.442} C_VEL
LIN {X 0,Y 418.135,Z 447.982,A -85,B 0,C 180,E1 -10180.899,E2 -10180.899} C_VEL
LIN {X 0,Y 418.708,Z 440.202,A -85,B 0,C 180,E1 -10182.11,E2 -10182.11} C_VEL
LIN {X 0,Y 419.395,Z 429.705,A -85,B 0,C 180,E1 -10183.434,E2 -10183.434} C_VEL
LIN {X 0,Y 420.261,Z 418.838,A -85,B 0,C 180,E1 -10184.526,E2 -10184.526} C_VEL
LIN {X 0,Y 421.11,Z 406.523,A -85,B 0,C 180,E1 -10185.486,E2 -10185.486} C_VEL
LIN {X 0,Y 421.881,Z 394.441,A -85,B 0,C 180,E1 -10186.201,E2 -10186.201} C_VEL
LIN {X 0,Y 422.473,Z 381.76,A -85,B 0,C 180,E1 -10186.737,E2 -10186.737} C_VEL
LIN {X 0,Y 422.933,Z 368.375,A -85,B 0,C 180,E1 -10187.091,E2 -10187.091} C_VEL
LIN {X 0,Y 423.717,Z 290.758,A -85,B 0,C 180,E1 -10188.449,E2 -10188.449} C_VEL
LIN {X 0,Y 419.83,Z 264.879,A -85,B 0,C 180,E1 -10189.125,E2 -10189.125} C_VEL
LIN {X 0,Y 419.538,Z 262.758,A -85,B 0,C 180,E1 -10189.192,E2 -10189.192} C_VEL
LIN {X 0,Y 420.783,Z 242.892,A -85,B 0,C 180,E1 -10192.954,E2 -10192.954} C_VEL
LIN {X 0,Y 421.307,Z 232.776,A -85,B 0,C 180,E1 -10194.9,E2 -10194.9} C_VEL
LIN {X 0,Y 418.842,Z 219.811,A -85,B 0,C 180,E1 -10197.593,E2 -10197.593} C_VEL
LIN {X 0,Y 418.356,Z 217.376,A -85,B 0,C 180,E1 -10198.125,E2 -10198.125} C_VEL
LIN {X 0,Y 418.209,Z 217.391,A -85,B 0,C 180,E1 -10201.395,E2 -10201.395} C_VEL
LIN {X 0,Y 418.261,Z 217.369,A -85,B 0,C 180,E1 -10204.579,E2 -10204.579} C_VEL
LIN {X 0,Y 418.216,Z 217.389,A -85,B 0,C 180,E1 -10207.831,E2 -10207.831} C_VEL
LIN {X 0,Y 418.204,Z 217.39,A -85,B 0,C 180,E1 -10210.949,E2 -10210.949} C_VEL
LIN {X 0,Y 418.202,Z 217.386,A -85,B 0,C 180,E1 -10213.728,E2 -10213.728} C_VEL
LIN {X 0,Y 418.195,Z 217.389,A -85,B 0,C 180,E1 -10216.447,E2 -10216.447} C_VEL
LIN {X 0,Y 418.201,Z 217.382,A -85,B 0,C 180,E1 -10219.132,E2 -10219.132} C_VEL
LIN {X 0,Y 418.231,Z 217.384,A -85,B 0,C 180,E1 -10222.775,E2 -10222.775} C_VEL
LIN {X 0,Y 418.24,Z 217.381,A -85,B 0,C 180,E1 -10226.322,E2 -10226.322} C_VEL
LIN {X 0,Y 418.233,Z 217.372,A -85,B 0,C 180,E1 -10229.727,E2 -10229.727} C_VEL
LIN {X 0,Y 418.201,Z 217.386,A -85,B 0,C 180,E1 -10233.016,E2 -10233.016} C_VEL
LIN {X 0,Y 418.247,Z 217.377,A -85,B 0,C 180,E1 -10236.216,E2 -10236.216} C_VEL
LIN {X 0,Y 418.239,Z 217.377,A -85,B 0,C 180,E1 -10239.337,E2 -10239.337} C_VEL
LIN {X 0,Y 418.268,Z 217.382,A -85,B 0,C 180,E1 -10242.395,E2 -10242.395} C_VEL
LIN {X 0,Y 418.276,Z 217.362,A -85,B 0,C 180,E1 -10245.402,E2 -10245.402} C_VEL
LIN {X 0,Y 418.302,Z 217.372,A -85,B 0,C 180,E1 -10248.369,E2 -10248.369} C_VEL
LIN {X 0,Y 418.367,Z 217.367,A -85,B 0,C 180,E1 -10251.304,E2 -10251.304} C_VEL
LIN {X 0,Y 418.456,Z 217.342,A -85,B 0,C 180,E1 -10254.217,E2 -10254.217} C_VEL
LIN {X 0,Y 418.53,Z 217.348,A -85,B 0,C 180,E1 -10258.076,E2 -10258.076} C_VEL
LIN {X 0,Y 418.471,Z 217.346,A -85,B 0,C 180,E1 -10260.963,E2 -10260.963} C_VEL
LIN {X 0,Y 418.469,Z 217.337,A -85,B 0,C 180,E1 -10262.888,E2 -10262.888} C_VEL
LIN {X 0,Y 418.475,Z 217.352,A -85,B 0,C 180,E1 -10266.643,E2 -10266.643} C_VEL
LIN {X 0,Y 418.331,Z 217.361,A -85,B 0,C 180,E1 -10269.672,E2 -10269.672} C_VEL
LIN {X 0,Y 418.338,Z 217.368,A -85,B 0,C 180,E1 -10273.001,E2 -10273.001} C_VEL
LIN {X 0,Y 418.304,Z 217.364,A -85,B 0,C 180,E1 -10276.736,E2 -10276.736} C_VEL
LIN {X 0,Y 418.263,Z 217.384,A -85,B 0,C 180,E1 -10279.791,E2 -10279.791} C_VEL
LIN {X 0,Y 418.231,Z 217.38,A -85,B 0,C 180,E1 -10282.737,E2 -10282.737} C_VEL
LIN {X 0,Y 418.264,Z 217.385,A -85,B 0,C 180,E1 -10285.905,E2 -10285.905} C_VEL
LIN {X 0,Y 418.258,Z 217.377,A -85,B 0,C 180,E1 -10289.163,E2 -10289.163} C_VEL
LIN {X 0,Y 418.252,Z 217.386,A -85,B 0,C 180,E1 -10292.845,E2 -10292.845} C_VEL
LIN {X 0,Y 418.243,Z 217.387,A -85,B 0,C 180,E1 -10296.24,E2 -10296.24} C_VEL
LIN {X 0,Y 418.251,Z 217.388,A -85,B 0,C 180,E1 -10299.683,E2 -10299.683} C_VEL
LIN {X 0,Y 418.227,Z 217.383,A -85,B 0,C 180,E1 -10302.323,E2 -10302.323} C_VEL
LIN {X 0,Y 418.238,Z 217.386,A -85,B 0,C 180,E1 -10305.111,E2 -10305.111} C_VEL
LIN {X 0,Y 418.239,Z 217.384,A -85,B 0,C 180,E1 -10307.768,E2 -10307.768} C_VEL
LIN {X 0,Y 418.253,Z 217.387,A -85,B 0,C 180,E1 -10310.62,E2 -10310.62} C_VEL
LIN {X 0,Y 418.241,Z 217.388,A -85,B 0,C 180,E1 -10313.977,E2 -10313.977} C_VEL
LIN {X 0,Y 418.3,Z 217.452,A -85,B 0,C 180,E1 -10315.884,E2 -10315.884} C_VEL
LIN {X 0,Y 419.913,Z 223.129,A -85,B 0,C 180,E1 -10316.539,E2 -10316.539} C_VEL
LIN {X 0,Y 421.596,Z 228.475,A -85,B 0,C 180,E1 -10316.732,E2 -10316.732} C_VEL
LIN {X 0,Y 424.902,Z 247.085,A -85,B 0,C 180,E1 -10317.25,E2 -10317.25} C_VEL
LIN {X 0,Y 423.662,Z 335.011,A -85,B 0,C 180,E1 -10318.777,E2 -10318.777} C_VEL
LIN {X 0,Y 423.291,Z 348.07,A -85,B 0,C 180,E1 -10319.18,E2 -10319.18} C_VEL
LIN {X 0,Y 422.828,Z 359.975,A -85,B 0,C 180,E1 -10319.735,E2 -10319.735} C_VEL
LIN {X 0,Y 422.245,Z 371.452,A -85,B 0,C 180,E1 -10320.458,E2 -10320.458} C_VEL
LIN {X 0,Y 421.46,Z 382.605,A -85,B 0,C 180,E1 -10321.354,E2 -10321.354} C_VEL
LIN {X 0,Y 420.661,Z 393.11,A -85,B 0,C 180,E1 -10322.417,E2 -10322.417} C_VEL
LIN {X 0,Y 419.863,Z 402.981,A -85,B 0,C 180,E1 -10323.669,E2 -10323.669} C_VEL
LIN {X 0,Y 419.168,Z 411.416,A -85,B 0,C 180,E1 -10324.987,E2 -10324.987} C_VEL
LIN {X 0,Y 418.534,Z 419.188,A -85,B 0,C 180,E1 -10326.498,E2 -10326.498} C_VEL
LIN {X 0,Y 418.062,Z 425.097,A -85,B 0,C 180,E1 -10327.937,E2 -10327.937} C_VEL
LIN {X 0,Y 417.673,Z 429.6,A -85,B 0,C 180,E1 -10329.308,E2 -10329.308} C_VEL
LIN {X 0,Y 417.462,Z 432.772,A -85,B 0,C 180,E1 -10330.523,E2 -10330.523} C_VEL
LIN {X 0,Y 417.152,Z 436.169,A -85,B 0,C 180,E1 -10332.348,E2 -10332.348} C_VEL
LIN {X 0,Y 417.043,Z 437.877,A -85,B 0,C 180,E1 -10333.858,E2 -10333.858} C_VEL
LIN {X 0,Y 416.953,Z 438.614,A -85,B 0,C 180,E1 -10335.356,E2 -10335.356} C_VEL
LIN {X 0,Y 416.982,Z 438.582,A -85,B 0,C 180,E1 -10336.353,E2 -10336.353} C_VEL
LIN {X 0,Y 417.064,Z 437.785,A -85,B 0,C 180,E1 -10337.789,E2 -10337.789} C_VEL
LIN {X 0,Y 417.089,Z 435.974,A -85,B 0,C 180,E1 -10339.32,E2 -10339.32} C_VEL
LIN {X 0,Y 417.242,Z 433.234,A -85,B 0,C 180,E1 -10340.793,E2 -10340.793} C_VEL
LIN {X 0,Y 417.447,Z 429.556,A -85,B 0,C 180,E1 -10342.23,E2 -10342.23} C_VEL
LIN {X 0,Y 416.924,Z 427.313,A -85,B 0,C 180,E1 -10342.976,E2 -10342.976} C_VEL
LIN {X 0,Y 414.333,Z 423.231,A -85,B 0,C 180,E1 -10344.169,E2 -10344.169} C_VEL
LIN {X 0,Y 411.76,Z 418.491,A -85,B 0,C 180,E1 -10345.327,E2 -10345.327} C_VEL
LIN {X 0,Y 411.273,Z 415.196,A -85,B 0,C 180,E1 -10346.009,E2 -10346.009} C_VEL
LIN {X 0,Y 411.795,Z 407.743,A -85,B 0,C 180,E1 -10347.311,E2 -10347.311} C_VEL
LIN {X 0,Y 412.376,Z 399.19,A -85,B 0,C 180,E1 -10348.536,E2 -10348.536} C_VEL
LIN {X 0,Y 413.118,Z 388.707,A -85,B 0,C 180,E1 -10349.757,E2 -10349.757} C_VEL
LIN {X 0,Y 413.827,Z 378.199,A -85,B 0,C 180,E1 -10350.731,E2 -10350.731} C_VEL
LIN {X 0,Y 414.45,Z 366.593,A -85,B 0,C 180,E1 -10351.58,E2 -10351.58} C_VEL
LIN {X 0,Y 414.925,Z 354.902,A -85,B 0,C 180,E1 -10352.236,E2 -10352.236} C_VEL
LIN {X 0,Y 415.326,Z 342.409,A -85,B 0,C 180,E1 -10352.735,E2 -10352.735} C_VEL
LIN {X 0,Y 415.523,Z 329.242,A -85,B 0,C 180,E1 -10353.063,E2 -10353.063} C_VEL
LIN {X 0,Y 416.42,Z 246.048,A -85,B 0,C 180,E1 -10354.497,E2 -10354.497} C_VEL
LIN {X 0,Y 412.368,Z 222.993,A -85,B 0,C 180,E1 -10355.073,E2 -10355.073} C_VEL
LIN {X 0,Y 411.477,Z 218.235,A -85,B 0,C 180,E1 -10355.637,E2 -10355.637} C_VEL
LIN {X 0,Y 411.419,Z 218.238,A -85,B 0,C 180,E1 -10357.856,E2 -10357.856} C_VEL
LIN {X 0,Y 411.288,Z 218.252,A -85,B 0,C 180,E1 -10361.834,E2 -10361.834} C_VEL
LIN {X 0,Y 411.264,Z 218.257,A -85,B 0,C 180,E1 -10364.854,E2 -10364.854} C_VEL
LIN {X 0,Y 411.257,Z 218.258,A -85,B 0,C 180,E1 -10367.916,E2 -10367.916} C_VEL
LIN {X 0,Y 411.203,Z 218.263,A -85,B 0,C 180,E1 -10371.035,E2 -10371.035} C_VEL
LIN {X 0,Y 411.197,Z 218.266,A -85,B 0,C 180,E1 -10374.218,E2 -10374.218} C_VEL
LIN {X 0,Y 411.155,Z 218.27,A -85,B 0,C 180,E1 -10377.486,E2 -10377.486} C_VEL
LIN {X 0,Y 411.202,Z 218.264,A -85,B 0,C 180,E1 -10379.714,E2 -10379.714} C_VEL
LIN {X 0,Y 411.211,Z 218.262,A -85,B 0,C 180,E1 -10383.157,E2 -10383.157} C_VEL
LIN {X 0,Y 411.196,Z 218.264,A -85,B 0,C 180,E1 -10386.552,E2 -10386.552} C_VEL
LIN {X 0,Y 411.169,Z 218.269,A -85,B 0,C 180,E1 -10389.72,E2 -10389.72} C_VEL
LIN {X 0,Y 411.166,Z 218.269,A -85,B 0,C 180,E1 -10393.136,E2 -10393.136} C_VEL
LIN {X 0,Y 411.168,Z 218.269,A -85,B 0,C 180,E1 -10395.882,E2 -10395.882} C_VEL
LIN {X 0,Y 411.161,Z 218.27,A -85,B 0,C 180,E1 -10399.493,E2 -10399.493} C_VEL
LIN {X 0,Y 411.181,Z 218.266,A -85,B 0,C 180,E1 -10402.024,E2 -10402.024} C_VEL
LIN {X 0,Y 411.194,Z 218.266,A -85,B 0,C 180,E1 -10405.127,E2 -10405.127} C_VEL
LIN {X 0,Y 411.159,Z 218.268,A -85,B 0,C 180,E1 -10408.002,E2 -10408.002} C_VEL
LIN {X 0,Y 411.173,Z 218.268,A -85,B 0,C 180,E1 -10411.406,E2 -10411.406} C_VEL
LIN {X 0,Y 411.193,Z 218.266,A -85,B 0,C 180,E1 -10414.941,E2 -10414.941} C_VEL
LIN {X 0,Y 411.251,Z 218.396,A -85,B 0,C 180,E1 -10417.669,E2 -10417.669} C_VEL
LIN {X 0,Y 412.58,Z 226.288,A -85,B 0,C 180,E1 -10419.691,E2 -10419.691} C_VEL
LIN {X 0,Y 412.607,Z 228.35,A -85,B 0,C 180,E1 -10420.196,E2 -10420.196} C_VEL
LIN {X 0,Y 416.229,Z 248.049,A -85,B 0,C 180,E1 -10420.776,E2 -10420.776} C_VEL
LIN {X 0,Y 414.522,Z 336.737,A -85,B 0,C 180,E1 -10422.676,E2 -10422.676} C_VEL
LIN {X 0,Y 414.156,Z 350.354,A -85,B 0,C 180,E1 -10423.169,E2 -10423.169} C_VEL
LIN {X 0,Y 413.774,Z 363.309,A -85,B 0,C 180,E1 -10423.851,E2 -10423.851} C_VEL
LIN {X 0,Y 413.136,Z 375.665,A -85,B 0,C 180,E1 -10424.711,E2 -10424.711} C_VEL
LIN {X 0,Y 412.578,Z 386.807,A -85,B 0,C 180,E1 -10425.7,E2 -10425.7} C_VEL
LIN {X 0,Y 412.089,Z 396.842,A -85,B 0,C 180,E1 -10426.808,E2 -10426.808} C_VEL
LIN {X 0,Y 411.524,Z 406.911,A -85,B 0,C 180,E1 -10428.174,E2 -10428.174} C_VEL
LIN {X 0,Y 411.047,Z 415.636,A -85,B 0,C 180,E1 -10429.658,E2 -10429.658} C_VEL
LIN {X 0,Y 410.656,Z 422.637,A -85,B 0,C 180,E1 -10431.139,E2 -10431.139} C_VEL
LIN {X 0,Y 410.397,Z 428.215,A -85,B 0,C 180,E1 -10432.62,E2 -10432.62} C_VEL
LIN {X 0,Y 410.241,Z 432.544,A -85,B 0,C 180,E1 -10434.1,E2 -10434.1} C_VEL
LIN {X 0,Y 410.167,Z 434.79,A -85,B 0,C 180,E1 -10435.085,E2 -10435.085} C_VEL
LIN {X 0,Y 410.092,Z 436.567,A -85,B 0,C 180,E1 -10436.069,E2 -10436.069} C_VEL
LIN {X 0,Y 410.144,Z 437.919,A -85,B 0,C 180,E1 -10437.053,E2 -10437.053} C_VEL
LIN {X 0,Y 410.057,Z 438.826,A -85,B 0,C 180,E1 -10438.035,E2 -10438.035} C_VEL
LIN {X 0,Y 409.999,Z 439.286,A -85,B 0,C 180,E1 -10439.018,E2 -10439.018} C_VEL
LIN {X 0,Y 410.017,Z 439.337,A -85,B 0,C 180,E1 -10440,E2 -10440} C_VEL
LIN {X 0,Y 410.069,Z 438.976,A -85,B 0,C 180,E1 -10440.982,E2 -10440.982} C_VEL
LIN {X 0,Y 410.151,Z 438.148,A -85,B 0,C 180,E1 -10441.964,E2 -10441.964} C_VEL
LIN {X 0,Y 410.311,Z 436.895,A -85,B 0,C 180,E1 -10442.945,E2 -10442.945} C_VEL
LIN {X 0,Y 410.539,Z 434.188,A -85,B 0,C 180,E1 -10444.418,E2 -10444.418} C_VEL
LIN {X 0,Y 410.623,Z 430.446,A -85,B 0,C 180,E1 -10445.894,E2 -10445.894} C_VEL
LIN {X 0,Y 411.233,Z 424.67,A -85,B 0,C 180,E1 -10447.59,E2 -10447.59} C_VEL
LIN {X 0,Y 411.699,Z 418.09,A -85,B 0,C 180,E1 -10449.085,E2 -10449.085} C_VEL
LIN {X 0,Y 412.427,Z 409.988,A -85,B 0,C 180,E1 -10450.555,E2 -10450.555} C_VEL
LIN {X 0,Y 413.1,Z 401.718,A -85,B 0,C 180,E1 -10451.78,E2 -10451.78} C_VEL
LIN {X 0,Y 413.716,Z 392.726,A -85,B 0,C 180,E1 -10452.883,E2 -10452.883} C_VEL
LIN {X 0,Y 414.625,Z 381.614,A -85,B 0,C 180,E1 -10453.977,E2 -10453.977} C_VEL
LIN {X 0,Y 415.357,Z 369.512,A -85,B 0,C 180,E1 -10454.931,E2 -10454.931} C_VEL
LIN {X 0,Y 416.017,Z 358.06,A -85,B 0,C 180,E1 -10455.621,E2 -10455.621} C_VEL
LIN {X 0,Y 416.497,Z 344.522,A -85,B 0,C 180,E1 -10456.229,E2 -10456.229} C_VEL
LIN {X 0,Y 416.888,Z 331.092,A -85,B 0,C 180,E1 -10456.622,E2 -10456.622} C_VEL
LIN {X 0,Y 419.249,Z 258.525,A -85,B 0,C 180,E1 -10458.341,E2 -10458.341} C_VEL
LIN {X 0,Y 419.365,Z 249.129,A -85,B 0,C 180,E1 -10458.589,E2 -10458.589} C_VEL
LIN {X 0,Y 416.896,Z 239.524,A -85,B 0,C 180,E1 -10459.041,E2 -10459.041} C_VEL
LIN {X 0,Y 414.292,Z 232.545,A -85,B 0,C 180,E1 -10459.466,E2 -10459.466} C_VEL
LIN {X 0,Y 413.138,Z 226.386,A -85,B 0,C 180,E1 -10461.453,E2 -10461.453} C_VEL
LIN {X 0,Y 411.235,Z 218.264,A -85,B 0,C 180,E1 -10464.322,E2 -10464.322} C_VEL
LIN {X 0,Y 411.265,Z 218.258,A -85,B 0,C 180,E1 -10467.477,E2 -10467.477} C_VEL
LIN {X 0,Y 411.195,Z 218.265,A -85,B 0,C 180,E1 -10470.847,E2 -10470.847} C_VEL
LIN {X 0,Y 411.211,Z 218.265,A -85,B 0,C 180,E1 -10474.333,E2 -10474.333} C_VEL
LIN {X 0,Y 411.199,Z 218.264,A -85,B 0,C 180,E1 -10477.973,E2 -10477.973} C_VEL
LIN {X 0,Y 411.186,Z 218.266,A -85,B 0,C 180,E1 -10480.504,E2 -10480.504} C_VEL
LIN {X 0,Y 411.178,Z 218.267,A -85,B 0,C 180,E1 -10483.133,E2 -10483.133} C_VEL
LIN {X 0,Y 411.172,Z 218.269,A -85,B 0,C 180,E1 -10485.881,E2 -10485.881} C_VEL
LIN {X 0,Y 411.165,Z 218.269,A -85,B 0,C 180,E1 -10488.772,E2 -10488.772} C_VEL
LIN {X 0,Y 411.194,Z 218.266,A -85,B 0,C 180,E1 -10492.025,E2 -10492.025} C_VEL
LIN {X 0,Y 411.21,Z 218.265,A -85,B 0,C 180,E1 -10495.666,E2 -10495.666} C_VEL
LIN {X 0,Y 411.216,Z 218.312,A -85,B 0,C 180,E1 -10498.99,E2 -10498.99} C_VEL
LIN {X 0,Y 413.508,Z 227.035,A -85,B 0,C 180,E1 -10501.582,E2 -10501.582} C_VEL
LIN {X 0,Y 415.364,Z 235.803,A -85,B 0,C 180,E1 -10503.9,E2 -10503.9} C_VEL
LIN {X 0,Y 415.784,Z 239.202,A -85,B 0,C 180,E1 -10504.734,E2 -10504.734} C_VEL
LIN {X 0,Y 414.249,Z 253.616,A -85,B 0,C 180,E1 -10507.821,E2 -10507.821} C_VEL
LIN {X 0,Y 413.556,Z 261.888,A -85,B 0,C 180,E1 -10509.516,E2 -10509.516} C_VEL
LIN {X 0,Y 417.087,Z 279.979,A -85,B 0,C 180,E1 -10510.276,E2 -10510.276} C_VEL
LIN {X 0,Y 418.55,Z 292.592,A -85,B 0,C 180,E1 -10510.716,E2 -10510.716} C_VEL
LIN {X 0,Y 416.262,Z 373.927,A -85,B 0,C 180,E1 -10512.655,E2 -10512.655} C_VEL
LIN {X 0,Y 415.634,Z 386.027,A -85,B 0,C 180,E1 -10513.104,E2 -10513.104} C_VEL
LIN {X 0,Y 414.787,Z 398.828,A -85,B 0,C 180,E1 -10513.764,E2 -10513.764} C_VEL
LIN {X 0,Y 413.962,Z 411.155,A -85,B 0,C 180,E1 -10514.616,E2 -10514.616} C_VEL
LIN {X 0,Y 413.098,Z 422.404,A -85,B 0,C 180,E1 -10515.592,E2 -10515.592} C_VEL
LIN {X 0,Y 412.211,Z 433.06,A -85,B 0,C 180,E1 -10516.747,E2 -10516.747} C_VEL
LIN {X 0,Y 411.557,Z 443.637,A -85,B 0,C 180,E1 -10518.174,E2 -10518.174} C_VEL
LIN {X 0,Y 410.86,Z 452.426,A -85,B 0,C 180,E1 -10519.652,E2 -10519.652} C_VEL
LIN {X 0,Y 410.447,Z 459.519,A -85,B 0,C 180,E1 -10521.134,E2 -10521.134} C_VEL
LIN {X 0,Y 410.175,Z 465.207,A -85,B 0,C 180,E1 -10522.616,E2 -10522.616} C_VEL
LIN {X 0,Y 409.995,Z 469.656,A -85,B 0,C 180,E1 -10524.096,E2 -10524.096} C_VEL
LIN {X 0,Y 410.013,Z 472.004,A -85,B 0,C 180,E1 -10525.082,E2 -10525.082} C_VEL
LIN {X 0,Y 409.94,Z 473.846,A -85,B 0,C 180,E1 -10526.067,E2 -10526.067} C_VEL
LIN {X 0,Y 409.968,Z 475.261,A -85,B 0,C 180,E1 -10527.051,E2 -10527.051} C_VEL
LIN {X 0,Y 410.018,Z 476.25,A -85,B 0,C 180,E1 -10528.034,E2 -10528.034} C_VEL
LIN {X 0,Y 409.98,Z 476.757,A -85,B 0,C 180,E1 -10529.017,E2 -10529.017} C_VEL
LIN {X 0,Y 409.986,Z 476.843,A -85,B 0,C 180,E1 -10529.999,E2 -10529.999} C_VEL
LIN {X 0,Y 409.98,Z 476.509,A -85,B 0,C 180,E1 -10530.981,E2 -10530.981} C_VEL
LIN {X 0,Y 410.022,Z 475.727,A -85,B 0,C 180,E1 -10531.963,E2 -10531.963} C_VEL
LIN {X 0,Y 410.028,Z 474.476,A -85,B 0,C 180,E1 -10532.946,E2 -10532.946} C_VEL
LIN {X 0,Y 410.005,Z 471.765,A -85,B 0,C 180,E1 -10534.423,E2 -10534.423} C_VEL
LIN {X 0,Y 410.041,Z 467.508,A -85,B 0,C 180,E1 -10536.223,E2 -10536.223} C_VEL
LIN {X 0,Y 410.26,Z 462.452,A -85,B 0,C 180,E1 -10537.876,E2 -10537.876} C_VEL
LIN {X 0,Y 410.604,Z 455.463,A -85,B 0,C 180,E1 -10539.606,E2 -10539.606} C_VEL
LIN {X 0,Y 411.139,Z 447.913,A -85,B 0,C 180,E1 -10541.086,E2 -10541.086} C_VEL
LIN {X 0,Y 411.75,Z 440.195,A -85,B 0,C 180,E1 -10542.318,E2 -10542.318} C_VEL
LIN {X 0,Y 412.424,Z 430.438,A -85,B 0,C 180,E1 -10543.587,E2 -10543.587} C_VEL
LIN {X 0,Y 413.394,Z 419.01,A -85,B 0,C 180,E1 -10544.773,E2 -10544.773} C_VEL
LIN {X 0,Y 414.21,Z 408.617,A -85,B 0,C 180,E1 -10545.625,E2 -10545.625} C_VEL
LIN {X 0,Y 415.034,Z 396.106,A -85,B 0,C 180,E1 -10546.413,E2 -10546.413} C_VEL
LIN {X 0,Y 415.692,Z 383.632,A -85,B 0,C 180,E1 -10546.987,E2 -10546.987} C_VEL
LIN {X 0,Y 416.221,Z 370.392,A -85,B 0,C 180,E1 -10547.376,E2 -10547.376} C_VEL
LIN {X 0,Y 417.097,Z 291.724,A -85,B 0,C 180,E1 -10548.783,E2 -10548.783} C_VEL
LIN {X 0,Y 413.482,Z 267.162,A -85,B 0,C 180,E1 -10549.434,E2 -10549.434} C_VEL
LIN {X 0,Y 412.631,Z 261.761,A -85,B 0,C 180,E1 -10549.594,E2 -10549.594} C_VEL
LIN {X 0,Y 413.952,Z 241.349,A -85,B 0,C 180,E1 -10553.537,E2 -10553.537} C_VEL
LIN {X 0,Y 414.37,Z 234.789,A -85,B 0,C 180,E1 -10554.819,E2 -10554.819} C_VEL
LIN {X 0,Y 412.697,Z 225.209,A -85,B 0,C 180,E1 -10556.825,E2 -10556.825} C_VEL
LIN {X 0,Y 411.306,Z 218.254,A -85,B 0,C 180,E1 -10558.338,E2 -10558.338} C_VEL
LIN {X 0,Y 411.162,Z 218.258,A -85,B 0,C 180,E1 -10561.996,E2 -10561.996} C_VEL
LIN {X 0,Y 411.206,Z 218.251,A -85,B 0,C 180,E1 -10564.877,E2 -10564.877} C_VEL
LIN {X 0,Y 411.189,Z 218.26,A -85,B 0,C 180,E1 -10568.166,E2 -10568.166} C_VEL
LIN {X 0,Y 411.163,Z 218.267,A -85,B 0,C 180,E1 -10571.805,E2 -10571.805} C_VEL
LIN {X 0,Y 411.168,Z 218.27,A -85,B 0,C 180,E1 -10575.508,E2 -10575.508} C_VEL
LIN {X 0,Y 411.141,Z 218.258,A -85,B 0,C 180,E1 -10578.773,E2 -10578.773} C_VEL
LIN {X 0,Y 411.179,Z 218.262,A -85,B 0,C 180,E1 -10582.025,E2 -10582.025} C_VEL
LIN {X 0,Y 411.197,Z 218.26,A -85,B 0,C 180,E1 -10585.666,E2 -10585.666} C_VEL
LIN {X 0,Y 411.18,Z 218.256,A -85,B 0,C 180,E1 -10589.152,E2 -10589.152} C_VEL
LIN {X 0,Y 411.167,Z 218.253,A -85,B 0,C 180,E1 -10591.406,E2 -10591.406} C_VEL
LIN {X 0,Y 411.178,Z 218.265,A -85,B 0,C 180,E1 -10594.941,E2 -10594.941} C_VEL
LIN {X 0,Y 411.193,Z 218.24,A -85,B 0,C 180,E1 -10597.913,E2 -10597.913} C_VEL
LIN {X 0,Y 411.209,Z 218.263,A -85,B 0,C 180,E1 -10601.051,E2 -10601.051} C_VEL
LIN {X 0,Y 411.233,Z 218.253,A -85,B 0,C 180,E1 -10604.131,E2 -10604.131} C_VEL
LIN {X 0,Y 411.294,Z 218.24,A -85,B 0,C 180,E1 -10607.166,E2 -10607.166} C_VEL
LIN {X 0,Y 411.279,Z 218.253,A -85,B 0,C 180,E1 -10610.161,E2 -10610.161} C_VEL
LIN {X 0,Y 411.376,Z 218.228,A -85,B 0,C 180,E1 -10613.132,E2 -10613.132} C_VEL
LIN {X 0,Y 411.28,Z 218.236,A -85,B 0,C 180,E1 -10615.099,E2 -10615.099} C_VEL
LIN {X 0,Y 411.499,Z 218.223,A -85,B 0,C 180,E1 -10618.043,E2 -10618.043} C_VEL
LIN {X 0,Y 411.435,Z 218.222,A -85,B 0,C 180,E1 -10620.979,E2 -10620.979} C_VEL
LIN {X 0,Y 411.427,Z 218.214,A -85,B 0,C 180,E1 -10622.938,E2 -10622.938} C_VEL
LIN {X 0,Y 411.437,Z 218.227,A -85,B 0,C 180,E1 -10626.645,E2 -10626.645} C_VEL
LIN {X 0,Y 411.283,Z 218.237,A -85,B 0,C 180,E1 -10629.839,E2 -10629.839} C_VEL
LIN {X 0,Y 411.297,Z 218.245,A -85,B 0,C 180,E1 -10633.105,E2 -10633.105} C_VEL
LIN {X 0,Y 411.249,Z 218.243,A -85,B 0,C 180,E1 -10636.889,E2 -10636.889} C_VEL
LIN {X 0,Y 411.223,Z 218.262,A -85,B 0,C 180,E1 -10639.988,E2 -10639.988} C_VEL
LIN {X 0,Y 411.196,Z 218.257,A -85,B 0,C 180,E1 -10643.148,E2 -10643.148} C_VEL
LIN {X 0,Y 411.232,Z 218.258,A -85,B 0,C 180,E1 -10646.382,E2 -10646.382} C_VEL
LIN {X 0,Y 411.194,Z 218.258,A -85,B 0,C 180,E1 -10649.714,E2 -10649.714} C_VEL
LIN {X 0,Y 411.201,Z 218.262,A -85,B 0,C 180,E1 -10653.157,E2 -10653.157} C_VEL
LIN {X 0,Y 411.19,Z 218.266,A -85,B 0,C 180,E1 -10656.554,E2 -10656.554} C_VEL
LIN {X 0,Y 411.214,Z 218.264,A -85,B 0,C 180,E1 -10659.73,E2 -10659.73} C_VEL
LIN {X 0,Y 411.173,Z 218.271,A -85,B 0,C 180,E1 -10663.134,E2 -10663.134} C_VEL
LIN {X 0,Y 411.17,Z 218.266,A -85,B 0,C 180,E1 -10665.881,E2 -10665.881} C_VEL
LIN {X 0,Y 411.162,Z 218.272,A -85,B 0,C 180,E1 -10668.773,E2 -10668.773} C_VEL
LIN {X 0,Y 411.204,Z 218.261,A -85,B 0,C 180,E1 -10671.833,E2 -10671.833} C_VEL
LIN {X 0,Y 411.261,Z 218.258,A -85,B 0,C 180,E1 -10675.542,E2 -10675.542} C_VEL
LIN {X 0,Y 412.679,Z 223.302,A -85,B 0,C 180,E1 -10676.122,E2 -10676.122} C_VEL
LIN {X 0,Y 415.157,Z 230.133,A -85,B 0,C 180,E1 -10676.395,E2 -10676.395} C_VEL
LIN {X 0,Y 418.281,Z 247.119,A -85,B 0,C 180,E1 -10676.886,E2 -10676.886} C_VEL
LIN {X 0,Y 416.984,Z 336.212,A -85,B 0,C 180,E1 -10678.467,E2 -10678.467} C_VEL
LIN {X 0,Y 416.578,Z 349.354,A -85,B 0,C 180,E1 -10678.893,E2 -10678.893} C_VEL
LIN {X 0,Y 416.011,Z 362.54,A -85,B 0,C 180,E1 -10679.55,E2 -10679.55} C_VEL
LIN {X 0,Y 415.353,Z 374.27,A -85,B 0,C 180,E1 -10680.337,E2 -10680.337} C_VEL
LIN {X 0,Y 414.41,Z 386.196,A -85,B 0,C 180,E1 -10681.375,E2 -10681.375} C_VEL
LIN {X 0,Y 413.57,Z 396.372,A -85,B 0,C 180,E1 -10682.494,E2 -10682.494} C_VEL
LIN {X 0,Y 412.831,Z 405.472,A -85,B 0,C 180,E1 -10683.73,E2 -10683.73} C_VEL
LIN {X 0,Y 412.093,Z 413.294,A -85,B 0,C 180,E1 -10685.034,E2 -10685.034} C_VEL
LIN {X 0,Y 411.437,Z 420.876,A -85,B 0,C 180,E1 -10686.601,E2 -10686.601} C_VEL
LIN {X 0,Y 411.021,Z 425.953,A -85,B 0,C 180,E1 -10687.904,E2 -10687.904} C_VEL
LIN {X 0,Y 410.593,Z 430.788,A -85,B 0,C 180,E1 -10689.459,E2 -10689.459} C_VEL
LIN {X 0,Y 410.299,Z 434.403,A -85,B 0,C 180,E1 -10691.008,E2 -10691.008} C_VEL
LIN {X 0,Y 410.107,Z 436.194,A -85,B 0,C 180,E1 -10692.034,E2 -10692.034} C_VEL
LIN {X 0,Y 409.971,Z 438.164,A -85,B 0,C 180,E1 -10693.74,E2 -10693.74} C_VEL
LIN {X 0,Y 409.891,Z 438.899,A -85,B 0,C 180,E1 -10695.098,E2 -10695.098} C_VEL
LIN {X 0,Y 409.873,Z 438.933,A -85,B 0,C 180,E1 -10696.111,E2 -10696.111} C_VEL
LIN {X 0,Y 409.962,Z 438.136,A -85,B 0,C 180,E1 -10697.732,E2 -10697.732} C_VEL
LIN {X 0,Y 410.007,Z 436.576,A -85,B 0,C 180,E1 -10699.133,E2 -10699.133} C_VEL
LIN {X 0,Y 410.125,Z 433.97,A -85,B 0,C 180,E1 -10700.632,E2 -10700.632} C_VEL
LIN {X 0,Y 410.38,Z 429.908,A -85,B 0,C 180,E1 -10702.275,E2 -10702.275} C_VEL
LIN {X 0,Y 410.664,Z 425.537,A -85,B 0,C 180,E1 -10703.629,E2 -10703.629} C_VEL
LIN {X 0,Y 411.001,Z 419.61,A -85,B 0,C 180,E1 -10705.096,E2 -10705.096} C_VEL
LIN {X 0,Y 411.273,Z 415.196,A -85,B 0,C 180,E1 -10706.009,E2 -10706.009} C_VEL
LIN {X 0,Y 410.807,Z 411.705,A -85,B 0,C 180,E1 -10706.673,E2 -10706.673} C_VEL
LIN {X 0,Y 408.371,Z 405.722,A -85,B 0,C 180,E1 -10707.728,E2 -10707.728} C_VEL
LIN {X 0,Y 406.049,Z 399.221,A -85,B 0,C 180,E1 -10708.726,E2 -10708.726} C_VEL
LIN {X 0,Y 405.756,Z 394.85,A -85,B 0,C 180,E1 -10709.289,E2 -10709.289} C_VEL
LIN {X 0,Y 406.466,Z 384.787,A -85,B 0,C 180,E1 -10710.373,E2 -10710.373} C_VEL
LIN {X 0,Y 407.186,Z 373.188,A -85,B 0,C 180,E1 -10711.361,E2 -10711.361} C_VEL
LIN {X 0,Y 407.79,Z 360.349,A -85,B 0,C 180,E1 -10712.201,E2 -10712.201} C_VEL
LIN {X 0,Y 408.262,Z 347.176,A -85,B 0,C 180,E1 -10712.816,E2 -10712.816} C_VEL
LIN {X 0,Y 408.607,Z 333.489,A -85,B 0,C 180,E1 -10713.229,E2 -10713.229} C_VEL
LIN {X 0,Y 409.685,Z 247.359,A -85,B 0,C 180,E1 -10714.742,E2 -10714.742} C_VEL
LIN {X 0,Y 405.525,Z 224.281,A -85,B 0,C 180,E1 -10715.33,E2 -10715.33} C_VEL
LIN {X 0,Y 405.115,Z 222.706,A -85,B 0,C 180,E1 -10715.414,E2 -10715.414} C_VEL
LIN {X 0,Y 404.439,Z 219.11,A -85,B 0,C 180,E1 -10715.829,E2 -10715.829} C_VEL
LIN {X 0,Y 404.271,Z 219.129,A -85,B 0,C 180,E1 -10719.003,E2 -10719.003} C_VEL
LIN {X 0,Y 404.261,Z 219.129,A -85,B 0,C 180,E1 -10722.042,E2 -10722.042} C_VEL
LIN {X 0,Y 404.21,Z 219.134,A -85,B 0,C 180,E1 -10725.119,E2 -10725.119} C_VEL
LIN {X 0,Y 404.215,Z 219.135,A -85,B 0,C 180,E1 -10728.239,E2 -10728.239} C_VEL
LIN {X 0,Y 404.145,Z 219.142,A -85,B 0,C 180,E1 -10731.42,E2 -10731.42} C_VEL
LIN {X 0,Y 404.142,Z 219.143,A -85,B 0,C 180,E1 -10734.669,E2 -10734.669} C_VEL
LIN {X 0,Y 404.112,Z 219.148,A -85,B 0,C 180,E1 -10738.007,E2 -10738.007} C_VEL
LIN {X 0,Y 404.149,Z 219.144,A -85,B 0,C 180,E1 -10740.286,E2 -10740.286} C_VEL
LIN {X 0,Y 404.144,Z 219.144,A -85,B 0,C 180,E1 -10743.813,E2 -10743.813} C_VEL
LIN {X 0,Y 404.138,Z 219.143,A -85,B 0,C 180,E1 -10746.874,E2 -10746.874} C_VEL
LIN {X 0,Y 404.123,Z 219.146,A -85,B 0,C 180,E1 -10750.075,E2 -10750.075} C_VEL
LIN {X 0,Y 404.146,Z 219.144,A -85,B 0,C 180,E1 -10753.082,E2 -10753.082} C_VEL
LIN {X 0,Y 404.125,Z 219.146,A -85,B 0,C 180,E1 -10755.922,E2 -10755.922} C_VEL
LIN {X 0,Y 404.106,Z 219.147,A -85,B 0,C 180,E1 -10758.633,E2 -10758.633} C_VEL
LIN {X 0,Y 404.138,Z 219.146,A -85,B 0,C 180,E1 -10761.496,E2 -10761.496} C_VEL
LIN {X 0,Y 404.165,Z 219.141,A -85,B 0,C 180,E1 -10764.981,E2 -10764.981} C_VEL
LIN {X 0,Y 404.14,Z 219.145,A -85,B 0,C 180,E1 -10767.378,E2 -10767.378} C_VEL
LIN {X 0,Y 404.153,Z 219.143,A -85,B 0,C 180,E1 -10770.862,E2 -10770.862} C_VEL
LIN {X 0,Y 404.157,Z 219.142,A -85,B 0,C 180,E1 -10774.723,E2 -10774.723} C_VEL
LIN {X 0,Y 404.186,Z 219.223,A -85,B 0,C 180,E1 -10777.509,E2 -10777.509} C_VEL
LIN {X 0,Y 405.513,Z 226.376,A -85,B 0,C 180,E1 -10779.373,E2 -10779.373} C_VEL
LIN {X 0,Y 405.612,Z 228.679,A -85,B 0,C 180,E1 -10779.95,E2 -10779.95} C_VEL
LIN {X 0,Y 409.302,Z 248.224,A -85,B 0,C 180,E1 -10780.535,E2 -10780.535} C_VEL
LIN {X 0,Y 407.558,Z 337.374,A -85,B 0,C 180,E1 -10782.5,E2 -10782.5} C_VEL
LIN {X 0,Y 407.196,Z 350.844,A -85,B 0,C 180,E1 -10783.002,E2 -10783.002} C_VEL
LIN {X 0,Y 406.782,Z 363.716,A -85,B 0,C 180,E1 -10783.695,E2 -10783.695} C_VEL
LIN {X 0,Y 406.128,Z 376.043,A -85,B 0,C 180,E1 -10784.57,E2 -10784.57} C_VEL
LIN {X 0,Y 405.557,Z 387.171,A -85,B 0,C 180,E1 -10785.575,E2 -10785.575} C_VEL
LIN {X 0,Y 405.014,Z 397.952,A -85,B 0,C 180,E1 -10786.796,E2 -10786.796} C_VEL
LIN {X 0,Y 404.54,Z 406.434,A -85,B 0,C 180,E1 -10787.967,E2 -10787.967} C_VEL
LIN {X 0,Y 404.033,Z 414.002,A -85,B 0,C 180,E1 -10789.222,E2 -10789.222} C_VEL
LIN {X 0,Y 403.686,Z 421.422,A -85,B 0,C 180,E1 -10790.733,E2 -10790.733} C_VEL
LIN {X 0,Y 403.327,Z 428.162,A -85,B 0,C 180,E1 -10792.49,E2 -10792.49} C_VEL
LIN {X 0,Y 403.161,Z 432.588,A -85,B 0,C 180,E1 -10793.996,E2 -10793.996} C_VEL
LIN {X 0,Y 403.106,Z 434.919,A -85,B 0,C 180,E1 -10794.999,E2 -10794.999} C_VEL
LIN {X 0,Y 403.006,Z 436.738,A -85,B 0,C 180,E1 -10796,E2 -10796} C_VEL
LIN {X 0,Y 403.044,Z 438.134,A -85,B 0,C 180,E1 -10797.001,E2 -10797.001} C_VEL
LIN {X 0,Y 402.988,Z 439.109,A -85,B 0,C 180,E1 -10798.001,E2 -10798.001} C_VEL
LIN {X 0,Y 402.924,Z 439.614,A -85,B 0,C 180,E1 -10799,E2 -10799} C_VEL
LIN {X 0,Y 402.937,Z 439.703,A -85,B 0,C 180,E1 -10800,E2 -10800} C_VEL
LIN {X 0,Y 402.991,Z 439.382,A -85,B 0,C 180,E1 -10800.999,E2 -10800.999} C_VEL
LIN {X 0,Y 403.08,Z 438.619,A -85,B 0,C 180,E1 -10801.998,E2 -10801.998} C_VEL
LIN {X 0,Y 403.248,Z 437.401,A -85,B 0,C 180,E1 -10802.997,E2 -10802.997} C_VEL
LIN {X 0,Y 403.499,Z 434.766,A -85,B 0,C 180,E1 -10804.495,E2 -10804.495} C_VEL
LIN {X 0,Y 403.589,Z 431.089,A -85,B 0,C 180,E1 -10805.997,E2 -10805.997} C_VEL
LIN {X 0,Y 404.247,Z 425.478,A -85,B 0,C 180,E1 -10807.7,E2 -10807.7} C_VEL
LIN {X 0,Y 404.751,Z 418.944,A -85,B 0,C 180,E1 -10809.242,E2 -10809.242} C_VEL
LIN {X 0,Y 405.523,Z 410.931,A -85,B 0,C 180,E1 -10810.737,E2 -10810.737} C_VEL
LIN {X 0,Y 406.228,Z 402.79,A -85,B 0,C 180,E1 -10811.982,E2 -10811.982} C_VEL
LIN {X 0,Y 407.045,Z 392.87,A -85,B 0,C 180,E1 -10813.225,E2 -10813.225} C_VEL
LIN {X 0,Y 407.992,Z 381.71,A -85,B 0,C 180,E1 -10814.337,E2 -10814.337} C_VEL
LIN {X 0,Y 408.678,Z 370.876,A -85,B 0,C 180,E1 -10815.211,E2 -10815.211} C_VEL
LIN {X 0,Y 409.407,Z 359.293,A -85,B 0,C 180,E1 -10815.942,E2 -10815.942} C_VEL
LIN {X 0,Y 409.914,Z 346.115,A -85,B 0,C 180,E1 -10816.561,E2 -10816.561} C_VEL
LIN {X 0,Y 410.358,Z 332.364,A -85,B 0,C 180,E1 -10816.991,E2 -10816.991} C_VEL
LIN {X 0,Y 412.969,Z 259.283,A -85,B 0,C 180,E1 -10818.779,E2 -10818.779} C_VEL
LIN {X 0,Y 413.11,Z 250.48,A -85,B 0,C 180,E1 -10819.019,E2 -10819.019} C_VEL
LIN {X 0,Y 410.701,Z 241.453,A -85,B 0,C 180,E1 -10819.473,E2 -10819.473} C_VEL
LIN {X 0,Y 407.365,Z 233.173,A -85,B 0,C 180,E1 -10820.016,E2 -10820.016} C_VEL
LIN {X 0,Y 405.495,Z 224.57,A -85,B 0,C 180,E1 -10822.97,E2 -10822.97} C_VEL
LIN {X 0,Y 404.209,Z 219.138,A -85,B 0,C 180,E1 -10825.048,E2 -10825.048} C_VEL
LIN {X 0,Y 404.201,Z 219.138,A -85,B 0,C 180,E1 -10827.999,E2 -10827.999} C_VEL
LIN {X 0,Y 404.145,Z 219.144,A -85,B 0,C 180,E1 -10831.557,E2 -10831.557} C_VEL
LIN {X 0,Y 404.19,Z 219.137,A -85,B 0,C 180,E1 -10835.016,E2 -10835.016} C_VEL
LIN {X 0,Y 404.159,Z 219.141,A -85,B 0,C 180,E1 -10838.756,E2 -10838.756} C_VEL
LIN {X 0,Y 404.128,Z 219.146,A -85,B 0,C 180,E1 -10841.599,E2 -10841.599} C_VEL
LIN {X 0,Y 404.15,Z 219.145,A -85,B 0,C 180,E1 -10844.521,E2 -10844.521} C_VEL
LIN {X 0,Y 404.137,Z 219.143,A -85,B 0,C 180,E1 -10847.294,E2 -10847.294} C_VEL
LIN {X 0,Y 404.158,Z 219.142,A -85,B 0,C 180,E1 -10849.953,E2 -10849.953} C_VEL
LIN {X 0,Y 404.139,Z 219.145,A -85,B 0,C 180,E1 -10853.125,E2 -10853.125} C_VEL
LIN {X 0,Y 404.149,Z 219.146,A -85,B 0,C 180,E1 -10856.187,E2 -10856.187} C_VEL
LIN {X 0,Y 404.162,Z 219.351,A -85,B 0,C 180,E1 -10858.321,E2 -10858.321} C_VEL
LIN {X 0,Y 406.249,Z 226.723,A -85,B 0,C 180,E1 -10860.672,E2 -10860.672} C_VEL
LIN {X 0,Y 408.371,Z 236.529,A -85,B 0,C 180,E1 -10863.418,E2 -10863.418} C_VEL
LIN {X 0,Y 409.037,Z 241.034,A -85,B 0,C 180,E1 -10864.56,E2 -10864.56} C_VEL
LIN {X 0,Y 407.415,Z 255.334,A -85,B 0,C 180,E1 -10867.696,E2 -10867.696} C_VEL
LIN {X 0,Y 406.871,Z 261.599,A -85,B 0,C 180,E1 -10868.981,E2 -10868.981} C_VEL
LIN {X 0,Y 410.314,Z 278.338,A -85,B 0,C 180,E1 -10869.739,E2 -10869.739} C_VEL
LIN {X 0,Y 412.158,Z 292.734,A -85,B 0,C 180,E1 -10870.28,E2 -10870.28} C_VEL
LIN {X 0,Y 409.993,Z 363.202,A -85,B 0,C 180,E1 -10871.995,E2 -10871.995} C_VEL
LIN {X 0,Y 409.496,Z 377.157,A -85,B 0,C 180,E1 -10872.392,E2 -10872.392} C_VEL
LIN {X 0,Y 408.775,Z 389.938,A -85,B 0,C 180,E1 -10872.94,E2 -10872.94} C_VEL
LIN {X 0,Y 407.907,Z 401.624,A -85,B 0,C 180,E1 -10873.611,E2 -10873.611} C_VEL
LIN {X 0,Y 407.002,Z 413.287,A -85,B 0,C 180,E1 -10874.474,E2 -10874.474} C_VEL
LIN {X 0,Y 406.035,Z 425.154,A -85,B 0,C 180,E1 -10875.592,E2 -10875.592} C_VEL
LIN {X 0,Y 405.176,Z 435.213,A -85,B 0,C 180,E1 -10876.762,E2 -10876.762} C_VEL
LIN {X 0,Y 404.608,Z 443.728,A -85,B 0,C 180,E1 -10877.968,E2 -10877.968} C_VEL
LIN {X 0,Y 403.827,Z 452.413,A -85,B 0,C 180,E1 -10879.47,E2 -10879.47} C_VEL
LIN {X 0,Y 403.406,Z 459.446,A -85,B 0,C 180,E1 -10880.978,E2 -10880.978} C_VEL
LIN {X 0,Y 403.123,Z 465.083,A -85,B 0,C 180,E1 -10882.486,E2 -10882.486} C_VEL
LIN {X 0,Y 402.919,Z 469.482,A -85,B 0,C 180,E1 -10883.992,E2 -10883.992} C_VEL
LIN {X 0,Y 402.921,Z 471.779,A -85,B 0,C 180,E1 -10884.996,E2 -10884.996} C_VEL
LIN {X 0,Y 402.859,Z 473.602,A -85,B 0,C 180,E1 -10885.997,E2 -10885.997} C_VEL
LIN {X 0,Y 402.866,Z 474.997,A -85,B 0,C 180,E1 -10886.999,E2 -10886.999} C_VEL
LIN {X 0,Y 402.946,Z 475.946,A -85,B 0,C 180,E1 -10888,E2 -10888} C_VEL
LIN {X 0,Y 402.905,Z 476.424,A -85,B 0,C 180,E1 -10888.999,E2 -10888.999} C_VEL
LIN {X 0,Y 402.908,Z 476.485,A -85,B 0,C 180,E1 -10889.999,E2 -10889.999} C_VEL
LIN {X 0,Y 402.905,Z 476.125,A -85,B 0,C 180,E1 -10890.998,E2 -10890.998} C_VEL
LIN {X 0,Y 402.953,Z 475.291,A -85,B 0,C 180,E1 -10891.998,E2 -10891.998} C_VEL
LIN {X 0,Y 402.929,Z 474.01,A -85,B 0,C 180,E1 -10892.998,E2 -10892.998} C_VEL
LIN {X 0,Y 402.915,Z 469.276,A -85,B 0,C 180,E1 -10895.504,E2 -10895.504} C_VEL
LIN {X 0,Y 403.034,Z 465.443,A -85,B 0,C 180,E1 -10897.01,E2 -10897.01} C_VEL
LIN {X 0,Y 403.281,Z 460.476,A -85,B 0,C 180,E1 -10898.517,E2 -10898.517} C_VEL
LIN {X 0,Y 403.658,Z 454.231,A -85,B 0,C 180,E1 -10900.026,E2 -10900.026} C_VEL
LIN {X 0,Y 404.253,Z 446.427,A -85,B 0,C 180,E1 -10901.532,E2 -10901.532} C_VEL
LIN {X 0,Y 405.11,Z 436.686,A -85,B 0,C 180,E1 -10903.033,E2 -10903.033} C_VEL
LIN {X 0,Y 405.796,Z 427.678,A -85,B 0,C 180,E1 -10904.159,E2 -10904.159} C_VEL
LIN {X 0,Y 406.79,Z 416.489,A -85,B 0,C 180,E1 -10905.275,E2 -10905.275} C_VEL
LIN {X 0,Y 407.636,Z 405.525,A -85,B 0,C 180,E1 -10906.14,E2 -10906.14} C_VEL
LIN {X 0,Y 408.412,Z 393.358,A -85,B 0,C 180,E1 -10906.88,E2 -10906.88} C_VEL
LIN {X 0,Y 409.141,Z 381.339,A -85,B 0,C 180,E1 -10907.396,E2 -10907.396} C_VEL
LIN {X 0,Y 409.601,Z 368.146,A -85,B 0,C 180,E1 -10907.763,E2 -10907.763} C_VEL
LIN {X 0,Y 410.461,Z 292.36,A -85,B 0,C 180,E1 -10909.136,E2 -10909.136} C_VEL
LIN {X 0,Y 407.032,Z 268.757,A -85,B 0,C 180,E1 -10909.777,E2 -10909.777} C_VEL
LIN {X 0,Y 405.727,Z 260.739,A -85,B 0,C 180,E1 -10910.014,E2 -10910.014} C_VEL
LIN {X 0,Y 407.123,Z 240.24,A -85,B 0,C 180,E1 -10914.049,E2 -10914.049} C_VEL
LIN {X 0,Y 407.359,Z 235.462,A -85,B 0,C 180,E1 -10915.003,E2 -10915.003} C_VEL
LIN {X 0,Y 405.334,Z 224.573,A -85,B 0,C 180,E1 -10917.327,E2 -10917.327} C_VEL
LIN {X 0,Y 404.255,Z 219.132,A -85,B 0,C 180,E1 -10918.559,E2 -10918.559} C_VEL
LIN {X 0,Y 404.137,Z 219.126,A -85,B 0,C 180,E1 -10922.62,E2 -10922.62} C_VEL
LIN {X 0,Y 404.176,Z 219.127,A -85,B 0,C 180,E1 -10925.189,E2 -10925.189} C_VEL
LIN {X 0,Y 404.129,Z 219.136,A -85,B 0,C 180,E1 -10928.758,E2 -10928.758} C_VEL
LIN {X 0,Y 404.108,Z 219.149,A -85,B 0,C 180,E1 -10931.597,E2 -10931.597} C_VEL
LIN {X 0,Y 404.139,Z 219.139,A -85,B 0,C 180,E1 -10934.521,E2 -10934.521} C_VEL
LIN {X 0,Y 404.117,Z 219.141,A -85,B 0,C 180,E1 -10937.293,E2 -10937.293} C_VEL
LIN {X 0,Y 404.125,Z 219.143,A -85,B 0,C 180,E1 -10939.95,E2 -10939.95} C_VEL
LIN {X 0,Y 404.127,Z 219.136,A -85,B 0,C 180,E1 -10943.125,E2 -10943.125} C_VEL
LIN {X 0,Y 404.137,Z 219.137,A -85,B 0,C 180,E1 -10946.187,E2 -10946.187} C_VEL
LIN {X 0,Y 404.135,Z 219.127,A -85,B 0,C 180,E1 -10949.714,E2 -10949.714} C_VEL
LIN {X 0,Y 404.095,Z 219.144,A -85,B 0,C 180,E1 -10953.116,E2 -10953.116} C_VEL
LIN {X 0,Y 404.139,Z 219.135,A -85,B 0,C 180,E1 -10956.424,E2 -10956.424} C_VEL
LIN {X 0,Y 404.182,Z 219.127,A -85,B 0,C 180,E1 -10959.874,E2 -10959.874} C_VEL
LIN {X 0,Y 404.207,Z 219.131,A -85,B 0,C 180,E1 -10962.993,E2 -10962.993} C_VEL
LIN {X 0,Y 404.274,Z 219.11,A -85,B 0,C 180,E1 -10966.939,E2 -10966.939} C_VEL
LIN {X 0,Y 404.245,Z 219.128,A -85,B 0,C 180,E1 -10969.988,E2 -10969.988} C_VEL
LIN {X 0,Y 404.327,Z 219.106,A -85,B 0,C 180,E1 -10973.011,E2 -10973.011} C_VEL
LIN {X 0,Y 404.25,Z 219.11,A -85,B 0,C 180,E1 -10975.013,E2 -10975.013} C_VEL
LIN {X 0,Y 404.468,Z 219.099,A -85,B 0,C 180,E1 -10978.009,E2 -10978.009} C_VEL
LIN {X 0,Y 404.399,Z 219.098,A -85,B 0,C 180,E1 -10980.996,E2 -10980.996} C_VEL
LIN {X 0,Y 404.387,Z 219.09,A -85,B 0,C 180,E1 -10982.989,E2 -10982.989} C_VEL
LIN {X 0,Y 404.383,Z 219.106,A -85,B 0,C 180,E1 -10986.645,E2 -10986.645} C_VEL
LIN {X 0,Y 404.282,Z 219.112,A -85,B 0,C 180,E1 -10989.001,E2 -10989.001} C_VEL
LIN {X 0,Y 404.247,Z 219.12,A -85,B 0,C 180,E1 -10992.042,E2 -10992.042} C_VEL
LIN {X 0,Y 404.198,Z 219.131,A -85,B 0,C 180,E1 -10995.119,E2 -10995.119} C_VEL
LIN {X 0,Y 404.197,Z 219.126,A -85,B 0,C 180,E1 -10998.239,E2 -10998.239} C_VEL
LIN {X 0,Y 404.153,Z 219.143,A -85,B 0,C 180,E1 -11001.419,E2 -11001.419} C_VEL
LIN {X 0,Y 404.17,Z 219.13,A -85,B 0,C 180,E1 -11004.666,E2 -11004.666} C_VEL
LIN {X 0,Y 404.189,Z 219.131,A -85,B 0,C 180,E1 -11008.001,E2 -11008.001} C_VEL
LIN {X 0,Y 404.134,Z 219.147,A -85,B 0,C 180,E1 -11011.559,E2 -11011.559} C_VEL
LIN {X 0,Y 404.18,Z 219.134,A -85,B 0,C 180,E1 -11015.017,E2 -11015.017} C_VEL
LIN {X 0,Y 404.155,Z 219.137,A -85,B 0,C 180,E1 -11018.758,E2 -11018.758} C_VEL
LIN {X 0,Y 404.12,Z 219.141,A -85,B 0,C 180,E1 -11021.601,E2 -11021.601} C_VEL
LIN {X 0,Y 404.146,Z 219.143,A -85,B 0,C 180,E1 -11024.524,E2 -11024.524} C_VEL
LIN {X 0,Y 404.136,Z 219.141,A -85,B 0,C 180,E1 -11027.297,E2 -11027.297} C_VEL
LIN {X 0,Y 404.166,Z 219.137,A -85,B 0,C 180,E1 -11029.957,E2 -11029.957} C_VEL
LIN {X 0,Y 404.135,Z 219.144,A -85,B 0,C 180,E1 -11033.126,E2 -11033.126} C_VEL
LIN {X 0,Y 404.191,Z 219.154,A -85,B 0,C 180,E1 -11035.19,E2 -11035.19} C_VEL
LIN {X 0,Y 405.583,Z 223.706,A -85,B 0,C 180,E1 -11035.699,E2 -11035.699} C_VEL
LIN {X 0,Y 408.779,Z 232.06,A -85,B 0,C 180,E1 -11036.053,E2 -11036.053} C_VEL
LIN {X 0,Y 411.736,Z 248.647,A -85,B 0,C 180,E1 -11036.54,E2 -11036.54} C_VEL
LIN {X 0,Y 410.368,Z 336.247,A -85,B 0,C 180,E1 -11038.115,E2 -11038.115} C_VEL
LIN {X 0,Y 409.939,Z 349.499,A -85,B 0,C 180,E1 -11038.547,E2 -11038.547} C_VEL
LIN {X 0,Y 409.346,Z 362.548,A -85,B 0,C 180,E1 -11039.202,E2 -11039.202} C_VEL
LIN {X 0,Y 408.684,Z 373.735,A -85,B 0,C 180,E1 -11039.956,E2 -11039.956} C_VEL
LIN {X 0,Y 407.859,Z 384.461,A -85,B 0,C 180,E1 -11040.872,E2 -11040.872} C_VEL
LIN {X 0,Y 406.881,Z 395.373,A -85,B 0,C 180,E1 -11042.053,E2 -11042.053} C_VEL
LIN {X 0,Y 406.071,Z 404.368,A -85,B 0,C 180,E1 -11043.258,E2 -11043.258} C_VEL
LIN {X 0,Y 405.275,Z 412.911,A -85,B 0,C 180,E1 -11044.664,E2 -11044.664} C_VEL
LIN {X 0,Y 404.564,Z 420.283,A -85,B 0,C 180,E1 -11046.179,E2 -11046.179} C_VEL
LIN {X 0,Y 404.081,Z 425.534,A -85,B 0,C 180,E1 -11047.504,E2 -11047.504} C_VEL
LIN {X 0,Y 403.611,Z 430.529,A -85,B 0,C 180,E1 -11049.087,E2 -11049.087} C_VEL
LIN {X 0,Y 403.274,Z 434.293,A -85,B 0,C 180,E1 -11050.664,E2 -11050.664} C_VEL
LIN {X 0,Y 403.072,Z 436.203,A -85,B 0,C 180,E1 -11051.71,E2 -11051.71} C_VEL
LIN {X 0,Y 402.906,Z 438.451,A -85,B 0,C 180,E1 -11053.615,E2 -11053.615} C_VEL
LIN {X 0,Y 402.814,Z 439.162,A -85,B 0,C 180,E1 -11054.83,E2 -11054.83} C_VEL
LIN {X 0,Y 402.795,Z 439.282,A -85,B 0,C 180,E1 -11055.862,E2 -11055.862} C_VEL
LIN {X 0,Y 402.895,Z 438.288,A -85,B 0,C 180,E1 -11057.918,E2 -11057.918} C_VEL
LIN {X 0,Y 402.914,Z 437.176,A -85,B 0,C 180,E1 -11058.939,E2 -11058.939} C_VEL
LIN {X 0,Y 402.939,Z 435.62,A -85,B 0,C 180,E1 -11059.956,E2 -11059.956} C_VEL
LIN {X 0,Y 403.189,Z 432.467,A -85,B 0,C 180,E1 -11061.481,E2 -11061.481} C_VEL
LIN {X 0,Y 403.492,Z 427.814,A -85,B 0,C 180,E1 -11063.136,E2 -11063.136} C_VEL
LIN {X 0,Y 403.738,Z 421.885,A -85,B 0,C 180,E1 -11064.758,E2 -11064.758} C_VEL
LIN {X 0,Y 404.303,Z 414.848,A -85,B 0,C 180,E1 -11066.264,E2 -11066.264} C_VEL
LIN {X 0,Y 404.954,Z 406.125,A -85,B 0,C 180,E1 -11067.763,E2 -11067.763} C_VEL
LIN {X 0,Y 405.558,Z 397.188,A -85,B 0,C 180,E1 -11069.008,E2 -11069.008} C_VEL
LIN {X 0,Y 405.756,Z 394.85,A -85,B 0,C 180,E1 -11069.289,E2 -11069.289} C_VEL
LIN {X 0,Y 405.46,Z 390.336,A -85,B 0,C 180,E1 -11069.826,E2 -11069.826} C_VEL
LIN {X 0,Y 403.161,Z 382.77,A -85,B 0,C 180,E1 -11070.678,E2 -11070.678} C_VEL
LIN {X 0,Y 400.854,Z 374.802,A -85,B 0,C 180,E1 -11071.456,E2 -11071.456} C_VEL
LIN {X 0,Y 400.524,Z 369.63,A -85,B 0,C 180,E1 -11071.859,E2 -11071.859} C_VEL
